LIN {X 0,Y 493.149,Z 1087.969,A -85,B 0,C 180,E1 23459.51,E2 23459.51} C_VEL
LIN {X 0,Y 495.56,Z 1076.918,A -85,B 0,C 180,E1 23456.854,E2 23456.854} C_VEL
LIN {X 0,Y 498.205,Z 1065.994,A -85,B 0,C 180,E1 23454.549,E2 23454.549} C_VEL
LIN {X 0,Y 501.969,Z 1051.472,A -85,B 0,C 180,E1 23451.868,E2 23451.868} C_VEL
LIN {X 0,Y 505.85,Z 1036.884,A -85,B 0,C 180,E1 23449.554,E2 23449.554} C_VEL
LIN {X 0,Y 509.727,Z 1022.712,A -85,B 0,C 180,E1 23447.563,E2 23447.563} C_VEL
LIN {X 0,Y 514.746,Z 1004.544,A -85,B 0,C 180,E1 23445.313,E2 23445.313} C_VEL
LIN {X 0,Y 519.682,Z 985.954,A -85,B 0,C 180,E1 23443.342,E2 23443.342} C_VEL
LIN {X 0,Y 524.249,Z 968.384,A -85,B 0,C 180,E1 23441.705,E2 23441.705} C_VEL
LIN {X 0,Y 529.619,Z 946.851,A -85,B 0,C 180,E1 23439.961,E2 23439.961} C_VEL
LIN {X 0,Y 534.306,Z 926.179,A -85,B 0,C 180,E1 23438.536,E2 23438.536} C_VEL
LIN {X 0,Y 538.281,Z 907.27,A -85,B 0,C 180,E1 23437.404,E2 23437.404} C_VEL
LIN {X 0,Y 542.76,Z 883.992,A -85,B 0,C 180,E1 23436.209,E2 23436.209} C_VEL
LIN {X 0,Y 546.654,Z 859.966,A -85,B 0,C 180,E1 23435.202,E2 23435.202} C_VEL
LIN {X 0,Y 549.579,Z 838.792,A -85,B 0,C 180,E1 23434.467,E2 23434.467} C_VEL
LIN {X 0,Y 552.455,Z 813.851,A -85,B 0,C 180,E1 23433.776,E2 23433.776} C_VEL
LIN {X 0,Y 554.553,Z 787.811,A -85,B 0,C 180,E1 23433.255,E2 23433.255} C_VEL
LIN {X 0,Y 565.206,Z 561.829,A -85,B 0,C 180,E1 23429.871,E2 23429.871} C_VEL
LIN {X 0,Y 571.63,Z 430.73,A -85,B 0,C 180,E1 23427.899,E2 23427.899} C_VEL
LIN {X 0,Y 561.962,Z 416.011,A -85,B 0,C 180,E1 23425.873,E2 23425.873} C_VEL
LIN {X 0,Y 552.616,Z 402.576,A -85,B 0,C 180,E1 23423.712,E2 23423.712} C_VEL
LIN {X 0,Y 543.559,Z 390.444,A -85,B 0,C 180,E1 23421.388,E2 23421.388} C_VEL
LIN {X 0,Y 535.724,Z 380.439,A -85,B 0,C 180,E1 23419.121,E2 23419.121} C_VEL
LIN {X 0,Y 531.614,Z 375.29,A -85,B 0,C 180,E1 23417.797,E2 23417.797} C_VEL
LIN {X 0,Y 527.184,Z 369.759,A -85,B 0,C 180,E1 23416.246,E2 23416.246} C_VEL
LIN {X 0,Y 522.155,Z 363.819,A -85,B 0,C 180,E1 23414.302,E2 23414.302} C_VEL
LIN {X 0,Y 517.658,Z 358.56,A -85,B 0,C 180,E1 23412.324,E2 23412.324} C_VEL
LIN {X 0,Y 512.757,Z 352.887,A -85,B 0,C 180,E1 23409.768,E2 23409.768} C_VEL
LIN {X 0,Y 508.771,Z 348.402,A -85,B 0,C 180,E1 23407.056,E2 23407.056} C_VEL
LIN {X 0,Y 508.042,Z 346.896,A -85,B 0,C 180,E1 23405.987,E2 23405.987} C_VEL
LIN {X 0,Y 505.565,Z 343.176,A -85,B 0,C 180,E1 23400.34,E2 23400.34} C_VEL
LIN {X 0,Y 505.432,Z 342.683,A -85,B 0,C 180,E1 23397.165,E2 23397.165} C_VEL
LIN {X 0,Y 505.943,Z 343.954,A -85,B 0,C 180,E1 23393.988,E2 23393.988} C_VEL
LIN {X 0,Y 508.736,Z 347.633,A -85,B 0,C 180,E1 23389.124,E2 23389.124} C_VEL
LIN {X 0,Y 510.625,Z 350.855,A -85,B 0,C 180,E1 23387.331,E2 23387.331} C_VEL
LIN {X 0,Y 514.02,Z 354.154,A -85,B 0,C 180,E1 23385.352,E2 23385.352} C_VEL
LIN {X 0,Y 519.518,Z 360.565,A -85,B 0,C 180,E1 23382.643,E2 23382.643} C_VEL
LIN {X 0,Y 524.302,Z 366.111,A -85,B 0,C 180,E1 23380.649,E2 23380.649} C_VEL
LIN {X 0,Y 528.297,Z 370.821,A -85,B 0,C 180,E1 23379.156,E2 23379.156} C_VEL
LIN {X 0,Y 534.627,Z 378.837,A -85,B 0,C 180,E1 23377.019,E2 23377.019} C_VEL
LIN {X 0,Y 541.875,Z 388.004,A -85,B 0,C 180,E1 23374.887,E2 23374.887} C_VEL
LIN {X 0,Y 549.446,Z 397.959,A -85,B 0,C 180,E1 23372.879,E2 23372.879} C_VEL
LIN {X 0,Y 559.137,Z 411.552,A -85,B 0,C 180,E1 23370.572,E2 23370.572} C_VEL
LIN {X 0,Y 568.555,Z 425.718,A -85,B 0,C 180,E1 23368.541,E2 23368.541} C_VEL
LIN {X 0,Y 574.364,Z 435.478,A -85,B 0,C 180,E1 23367.361,E2 23367.361} C_VEL
LIN {X 0,Y 564.405,Z 645.919,A -85,B 0,C 180,E1 23364.13,E2 23364.13} C_VEL
LIN {X 0,Y 556.556,Z 821.444,A -85,B 0,C 180,E1 23361.46,E2 23361.46} C_VEL
LIN {X 0,Y 554.253,Z 849.077,A -85,B 0,C 180,E1 23360.931,E2 23360.931} C_VEL
LIN {X 0,Y 551.182,Z 874.995,A -85,B 0,C 180,E1 23360.252,E2 23360.252} C_VEL
LIN {X 0,Y 548.203,Z 896.474,A -85,B 0,C 180,E1 23359.554,E2 23359.554} C_VEL
LIN {X 0,Y 544.933,Z 917.274,A -85,B 0,C 180,E1 23358.748,E2 23358.748} C_VEL
LIN {X 0,Y 540.875,Z 940.581,A -85,B 0,C 180,E1 23357.684,E2 23357.684} C_VEL
LIN {X 0,Y 535.726,Z 966.965,A -85,B 0,C 180,E1 23356.243,E2 23356.243} C_VEL
LIN {X 0,Y 531.462,Z 987.244,A -85,B 0,C 180,E1 23354.954,E2 23354.954} C_VEL
LIN {X 0,Y 527.075,Z 1007.137,A -85,B 0,C 180,E1 23353.52,E2 23353.52} C_VEL
LIN {X 0,Y 521.899,Z 1029.99,A -85,B 0,C 180,E1 23351.652,E2 23351.652} C_VEL
LIN {X 0,Y 516.787,Z 1051.566,A -85,B 0,C 180,E1 23349.606,E2 23349.606} C_VEL
LIN {X 0,Y 512.688,Z 1068.925,A -85,B 0,C 180,E1 23347.761,E2 23347.761} C_VEL
LIN {X 0,Y 508.88,Z 1085.197,A -85,B 0,C 180,E1 23345.84,E2 23345.84} C_VEL
LIN {X 0,Y 504.662,Z 1103.524,A -85,B 0,C 180,E1 23343.421,E2 23343.421} C_VEL
LIN {X 0,Y 500.671,Z 1121.052,A -85,B 0,C 180,E1 23340.747,E2 23340.747} C_VEL
LIN {X 0,Y 497.946,Z 1133.879,A -85,B 0,C 180,E1 23338.548,E2 23338.548} C_VEL
LIN {X 0,Y 495.478,Z 1146.019,A -85,B 0,C 180,E1 23336.227,E2 23336.227} C_VEL
LIN {X 0,Y 493.194,Z 1158.493,A -85,B 0,C 180,E1 23333.54,E2 23333.54} C_VEL
LIN {X 0,Y 491.411,Z 1169.048,A -85,B 0,C 180,E1 23330.859,E2 23330.859} C_VEL
LIN {X 0,Y 489.941,Z 1178.442,A -85,B 0,C 180,E1 23327.948,E2 23327.948} C_VEL
LIN {X 0,Y 489.053,Z 1185.745,A -85,B 0,C 180,E1 23325.292,E2 23325.292} C_VEL
LIN {X 0,Y 488.48,Z 1191.567,A -85,B 0,C 180,E1 23322.772,E2 23322.772} C_VEL
LIN {X 0,Y 488.152,Z 1196.51,A -85,B 0,C 180,E1 23320.146,E2 23320.146} C_VEL
LIN {X 0,Y 487.972,Z 1200.927,A -85,B 0,C 180,E1 23317.062,E2 23317.062} C_VEL
LIN {X 0,Y 487.915,Z 1203.615,A -85,B 0,C 180,E1 23313.995,E2 23313.995} C_VEL
LIN {X 0,Y 487.912,Z 1204.735,A -85,B 0,C 180,E1 23311.409,E2 23311.409} C_VEL
LIN {X 0,Y 487.906,Z 1204.825,A -85,B 0,C 180,E1 23309.061,E2 23309.061} C_VEL
LIN {X 0,Y 487.915,Z 1203.955,A -85,B 0,C 180,E1 23306.593,E2 23306.593} C_VEL
LIN {X 0,Y 487.942,Z 1202.076,A -85,B 0,C 180,E1 23304.119,E2 23304.119} C_VEL
LIN {X 0,Y 488.027,Z 1199.188,A -85,B 0,C 180,E1 23301.636,E2 23301.636} C_VEL
LIN {X 0,Y 488.216,Z 1195.271,A -85,B 0,C 180,E1 23299.14,E2 23299.14} C_VEL
LIN {X 0,Y 488.681,Z 1189.532,A -85,B 0,C 180,E1 23296.271,E2 23296.271} C_VEL
LIN {X 0,Y 489.58,Z 1181.265,A -85,B 0,C 180,E1 23293.02,E2 23293.02} C_VEL
LIN {X 0,Y 490.735,Z 1173.099,A -85,B 0,C 180,E1 23290.356,E2 23290.356} C_VEL
LIN {X 0,Y 492.077,Z 1164.967,A -85,B 0,C 180,E1 23288.045,E2 23288.045} C_VEL
LIN {X 0,Y 493.665,Z 1155.796,A -85,B 0,C 180,E1 23285.85,E2 23285.85} C_VEL
LIN {X 0,Y 495.728,Z 1144.888,A -85,B 0,C 180,E1 23283.529,E2 23283.529} C_VEL
LIN {X 0,Y 498.377,Z 1132.01,A -85,B 0,C 180,E1 23281.086,E2 23281.086} C_VEL
LIN {X 0,Y 502.265,Z 1114.42,A -85,B 0,C 180,E1 23278.161,E2 23278.161} C_VEL
LIN {X 0,Y 505.899,Z 1098.541,A -85,B 0,C 180,E1 23275.855,E2 23275.855} C_VEL
LIN {X 0,Y 509.534,Z 1083.124,A -85,B 0,C 180,E1 23273.848,E2 23273.848} C_VEL
LIN {X 0,Y 513.567,Z 1066.164,A -85,B 0,C 180,E1 23271.866,E2 23271.866} C_VEL
LIN {X 0,Y 518.894,Z 1043.729,A -85,B 0,C 180,E1 23269.566,E2 23269.566} C_VEL
LIN {X 0,Y 523.308,Z 1024.462,A -85,B 0,C 180,E1 23267.847,E2 23267.847} C_VEL
LIN {X 0,Y 527.446,Z 1005.817,A -85,B 0,C 180,E1 23266.369,E2 23266.369} C_VEL
LIN {X 0,Y 531.6,Z 986.265,A -85,B 0,C 180,E1 23264.993,E2 23264.993} C_VEL
LIN {X 0,Y 536.616,Z 961.242,A -85,B 0,C 180,E1 23263.462,E2 23263.462} C_VEL
LIN {X 0,Y 540.86,Z 937.419,A -85,B 0,C 180,E1 23262.236,E2 23262.236} C_VEL
LIN {X 0,Y 544.215,Z 916.811,A -85,B 0,C 180,E1 23261.325,E2 23261.325} C_VEL
LIN {X 0,Y 547.287,Z 895.889,A -85,B 0,C 180,E1 23260.536,E2 23260.536} C_VEL
LIN {X 0,Y 550.407,Z 871.646,A -85,B 0,C 180,E1 23259.775,E2 23259.775} C_VEL
LIN {X 0,Y 553.269,Z 843.484,A -85,B 0,C 180,E1 23259.097,E2 23259.097} C_VEL
LIN {X 0,Y 554.958,Z 820.18,A -85,B 0,C 180,E1 23258.674,E2 23258.674} C_VEL
LIN {X 0,Y 562.927,Z 611.986,A -85,B 0,C 180,E1 23255.596,E2 23255.596} C_VEL
LIN {X 0,Y 569.954,Z 434.455,A -85,B 0,C 180,E1 23252.946,E2 23252.946} C_VEL
LIN {X 0,Y 553.295,Z 409.736,A -85,B 0,C 180,E1 23250.158,E2 23250.158} C_VEL
LIN {X 0,Y 539.586,Z 390.209,A -85,B 0,C 180,E1 23247.628,E2 23247.628} C_VEL
LIN {X 0,Y 527.933,Z 374.572,A -85,B 0,C 180,E1 23245.253,E2 23245.253} C_VEL
LIN {X 0,Y 517.455,Z 360.976,A -85,B 0,C 180,E1 23242.915,E2 23242.915} C_VEL
LIN {X 0,Y 511.897,Z 354.221,A -85,B 0,C 180,E1 23241.575,E2 23241.575} C_VEL
LIN {X 0,Y 507.878,Z 349.051,A -85,B 0,C 180,E1 23240.514,E2 23240.514} C_VEL
LIN {X 0,Y 505.11,Z 344.247,A -85,B 0,C 180,E1 23239.184,E2 23239.184} C_VEL
LIN {X 0,Y 502.34,Z 339.33,A -85,B 0,C 180,E1 23237.731,E2 23237.731} C_VEL
LIN {X 0,Y 500.084,Z 335.455,A -85,B 0,C 180,E1 23236.494,E2 23236.494} C_VEL
LIN {X 0,Y 499.057,Z 333.831,A -85,B 0,C 180,E1 23235.932,E2 23235.932} C_VEL
LIN {X 0,Y 496.972,Z 330.249,A -85,B 0,C 180,E1 23234.685,E2 23234.685} C_VEL
LIN {X 0,Y 496.045,Z 328.722,A -85,B 0,C 180,E1 23234.117,E2 23234.117} C_VEL
LIN {X 0,Y 493.83,Z 325.381,A -85,B 0,C 180,E1 23232.75,E2 23232.75} C_VEL
LIN {X 0,Y 492.938,Z 323.506,A -85,B 0,C 180,E1 23232.06,E2 23232.06} C_VEL
LIN {X 0,Y 490.401,Z 319.891,A -85,B 0,C 180,E1 23230.336,E2 23230.336} C_VEL
LIN {X 0,Y 490.011,Z 318.347,A -85,B 0,C 180,E1 23229.632,E2 23229.632} C_VEL
LIN {X 0,Y 489.975,Z 318.197,A -85,B 0,C 180,E1 23226.327,E2 23226.327} C_VEL
LIN {X 0,Y 489.984,Z 318.197,A -85,B 0,C 180,E1 23222.69,E2 23222.69} C_VEL
LIN {X 0,Y 489.988,Z 318.196,A -85,B 0,C 180,E1 23219.11,E2 23219.11} C_VEL
LIN {X 0,Y 489.979,Z 318.198,A -85,B 0,C 180,E1 23215.552,E2 23215.552} C_VEL
LIN {X 0,Y 489.968,Z 318.2,A -85,B 0,C 180,E1 23212.023,E2 23212.023} C_VEL
LIN {X 0,Y 489.987,Z 318.199,A -85,B 0,C 180,E1 23208.464,E2 23208.464} C_VEL
LIN {X 0,Y 489.996,Z 318.196,A -85,B 0,C 180,E1 23204.835,E2 23204.835} C_VEL
LIN {X 0,Y 489.973,Z 318.196,A -85,B 0,C 180,E1 23201.236,E2 23201.236} C_VEL
LIN {X 0,Y 489.962,Z 318.184,A -85,B 0,C 180,E1 23197.692,E2 23197.692} C_VEL
LIN {X 0,Y 490.031,Z 318.559,A -85,B 0,C 180,E1 23195.915,E2 23195.915} C_VEL
LIN {X 0,Y 491.731,Z 322.184,A -85,B 0,C 180,E1 23194.334,E2 23194.334} C_VEL
LIN {X 0,Y 493.389,Z 324.398,A -85,B 0,C 180,E1 23193.263,E2 23193.263} C_VEL
LIN {X 0,Y 495.592,Z 328.394,A -85,B 0,C 180,E1 23191.697,E2 23191.697} C_VEL
LIN {X 0,Y 496.572,Z 329.857,A -85,B 0,C 180,E1 23191.101,E2 23191.101} C_VEL
LIN {X 0,Y 498.866,Z 333.836,A -85,B 0,C 180,E1 23189.663,E2 23189.663} C_VEL
LIN {X 0,Y 502.443,Z 340.404,A -85,B 0,C 180,E1 23187.539,E2 23187.539} C_VEL
LIN {X 0,Y 505.203,Z 345.524,A -85,B 0,C 180,E1 23186.022,E2 23186.022} C_VEL
LIN {X 0,Y 507.222,Z 348.663,A -85,B 0,C 180,E1 23185.201,E2 23185.201} C_VEL
LIN {X 0,Y 513.433,Z 356.368,A -85,B 0,C 180,E1 23183.629,E2 23183.629} C_VEL
LIN {X 0,Y 523.089,Z 368.663,A -85,B 0,C 180,E1 23181.383,E2 23181.383} C_VEL
LIN {X 0,Y 533.138,Z 382.053,A -85,B 0,C 180,E1 23179.259,E2 23179.259} C_VEL
LIN {X 0,Y 545.23,Z 398.991,A -85,B 0,C 180,E1 23176.912,E2 23176.912} C_VEL
LIN {X 0,Y 559.529,Z 420.202,A -85,B 0,C 180,E1 23174.39,E2 23174.39} C_VEL
LIN {X 0,Y 564.66,Z 428.424,A -85,B 0,C 180,E1 23173.534,E2 23173.534} C_VEL
LIN {X 0,Y 555.474,Z 654.275,A -85,B 0,C 180,E1 23170.226,E2 23170.226} C_VEL
LIN {X 0,Y 550.131,Z 787.111,A -85,B 0,C 180,E1 23168.273,E2 23168.273} C_VEL
LIN {X 0,Y 548.159,Z 813.65,A -85,B 0,C 180,E1 23167.744,E2 23167.744} C_VEL
LIN {X 0,Y 545.611,Z 837.887,A -85,B 0,C 180,E1 23167.078,E2 23167.078} C_VEL
LIN {X 0,Y 543.174,Z 857.409,A -85,B 0,C 180,E1 23166.414,E2 23166.414} C_VEL
LIN {X 0,Y 541.449,Z 864.935,A -85,B 0,C 180,E1 23166.216,E2 23166.216} C_VEL
LIN {X 0,Y 534.335,Z 883.517,A -85,B 0,C 180,E1 23165.889,E2 23165.889} C_VEL
LIN {X 0,Y 532.422,Z 890.42,A -85,B 0,C 180,E1 23165.628,E2 23165.628} C_VEL
LIN {X 0,Y 528.887,Z 909.703,A -85,B 0,C 180,E1 23164.617,E2 23164.617} C_VEL
LIN {X 0,Y 524.361,Z 932.228,A -85,B 0,C 180,E1 23163.244,E2 23163.244} C_VEL
LIN {X 0,Y 519.531,Z 953.612,A -85,B 0,C 180,E1 23161.695,E2 23161.695} C_VEL
LIN {X 0,Y 515.319,Z 971.28,A -85,B 0,C 180,E1 23160.232,E2 23160.232} C_VEL
LIN {X 0,Y 510.276,Z 991.608,A -85,B 0,C 180,E1 23158.306,E2 23158.306} C_VEL
LIN {X 0,Y 505.499,Z 1009.737,A -85,B 0,C 180,E1 23156.299,E2 23156.299} C_VEL
LIN {X 0,Y 501.644,Z 1024.173,A -85,B 0,C 180,E1 23154.493,E2 23154.493} C_VEL
LIN {X 0,Y 497.358,Z 1040.344,A -85,B 0,C 180,E1 23152.206,E2 23152.206} C_VEL
LIN {X 0,Y 493.255,Z 1055.784,A -85,B 0,C 180,E1 23149.663,E2 23149.663} C_VEL
LIN {X 0,Y 490.261,Z 1067.568,A -85,B 0,C 180,E1 23147.445,E2 23147.445} C_VEL
LIN {X 0,Y 487.453,Z 1079.24,A -85,B 0,C 180,E1 23144.951,E2 23144.951} C_VEL
LIN {X 0,Y 484.785,Z 1091.351,A -85,B 0,C 180,E1 23141.902,E2 23141.902} C_VEL
LIN {X 0,Y 483.145,Z 1099.766,A -85,B 0,C 180,E1 23139.409,E2 23139.409} C_VEL
LIN {X 0,Y 481.86,Z 1107.651,A -85,B 0,C 180,E1 23136.673,E2 23136.673} C_VEL
LIN {X 0,Y 480.875,Z 1115.108,A -85,B 0,C 180,E1 23133.457,E2 23133.457} C_VEL
LIN {X 0,Y 480.406,Z 1119.686,A -85,B 0,C 180,E1 23130.954,E2 23130.954} C_VEL
LIN {X 0,Y 480.182,Z 1123.237,A -85,B 0,C 180,E1 23128.449,E2 23128.449} C_VEL
LIN {X 0,Y 480.051,Z 1126.112,A -85,B 0,C 180,E1 23125.58,E2 23125.58} C_VEL
LIN {X 0,Y 480.017,Z 1127.597,A -85,B 0,C 180,E1 23122.536,E2 23122.536} C_VEL
LIN {X 0,Y 480.009,Z 1127.73,A -85,B 0,C 180,E1 23120.044,E2 23120.044} C_VEL
LIN {X 0,Y 480.042,Z 1126.911,A -85,B 0,C 180,E1 23117.612,E2 23117.612} C_VEL
LIN {X 0,Y 480.092,Z 1125.029,A -85,B 0,C 180,E1 23115.034,E2 23115.034} C_VEL
LIN {X 0,Y 480.33,Z 1121.374,A -85,B 0,C 180,E1 23111.931,E2 23111.931} C_VEL
LIN {X 0,Y 480.725,Z 1116.685,A -85,B 0,C 180,E1 23109.166,E2 23109.166} C_VEL
LIN {X 0,Y 481.392,Z 1111.294,A -85,B 0,C 180,E1 23106.627,E2 23106.627} C_VEL
LIN {X 0,Y 482.54,Z 1104.025,A -85,B 0,C 180,E1 23103.798,E2 23103.798} C_VEL
LIN {X 0,Y 484.362,Z 1094.295,A -85,B 0,C 180,E1 23100.71,E2 23100.71} C_VEL
LIN {X 0,Y 486.355,Z 1085.178,A -85,B 0,C 180,E1 23098.245,E2 23098.245} C_VEL
LIN {X 0,Y 489.044,Z 1074.172,A -85,B 0,C 180,E1 23095.647,E2 23095.647} C_VEL
LIN {X 0,Y 492.766,Z 1060.042,A -85,B 0,C 180,E1 23092.795,E2 23092.795} C_VEL
LIN {X 0,Y 496.209,Z 1047.557,A -85,B 0,C 180,E1 23090.6,E2 23090.6} C_VEL
LIN {X 0,Y 500.308,Z 1033.218,A -85,B 0,C 180,E1 23088.371,E2 23088.371} C_VEL
LIN {X 0,Y 505.662,Z 1014.624,A -85,B 0,C 180,E1 23085.873,E2 23085.873} C_VEL
LIN {X 0,Y 509.914,Z 999.653,A -85,B 0,C 180,E1 23084.117,E2 23084.117} C_VEL
LIN {X 0,Y 514.514,Z 983.146,A -85,B 0,C 180,E1 23082.4,E2 23082.4} C_VEL
LIN {X 0,Y 520.076,Z 962.549,A -85,B 0,C 180,E1 23080.529,E2 23080.529} C_VEL
LIN {X 0,Y 525.106,Z 942.324,A -85,B 0,C 180,E1 23078.962,E2 23078.962} C_VEL
LIN {X 0,Y 529.206,Z 924.828,A -85,B 0,C 180,E1 23077.776,E2 23077.776} C_VEL
LIN {X 0,Y 533.347,Z 905.742,A -85,B 0,C 180,E1 23076.643,E2 23076.643} C_VEL
LIN {X 0,Y 538.141,Z 881.083,A -85,B 0,C 180,E1 23075.405,E2 23075.405} C_VEL
LIN {X 0,Y 541.68,Z 859.732,A -85,B 0,C 180,E1 23074.52,E2 23074.52} C_VEL
LIN {X 0,Y 544.703,Z 838.45,A -85,B 0,C 180,E1 23073.786,E2 23073.786} C_VEL
LIN {X 0,Y 547.724,Z 812.789,A -85,B 0,C 180,E1 23073.081,E2 23073.081} C_VEL
LIN {X 0,Y 549.775,Z 787.528,A -85,B 0,C 180,E1 23072.582,E2 23072.582} C_VEL
LIN {X 0,Y 561.031,Z 557.477,A -85,B 0,C 180,E1 23069.121,E2 23069.121} C_VEL
LIN {X 0,Y 567.259,Z 435.24,A -85,B 0,C 180,E1 23067.277,E2 23067.277} C_VEL
LIN {X 0,Y 558.135,Z 421.099,A -85,B 0,C 180,E1 23065.295,E2 23065.295} C_VEL
LIN {X 0,Y 548.312,Z 407.108,A -85,B 0,C 180,E1 23062.942,E2 23062.942} C_VEL
LIN {X 0,Y 540.587,Z 396.703,A -85,B 0,C 180,E1 23060.887,E2 23060.887} C_VEL
LIN {X 0,Y 533.593,Z 387.597,A -85,B 0,C 180,E1 23058.803,E2 23058.803} C_VEL
LIN {X 0,Y 529.702,Z 382.655,A -85,B 0,C 180,E1 23057.523,E2 23057.523} C_VEL
LIN {X 0,Y 525.337,Z 377.159,A -85,B 0,C 180,E1 23055.964,E2 23055.964} C_VEL
LIN {X 0,Y 520.538,Z 371.373,A -85,B 0,C 180,E1 23054.069,E2 23054.069} C_VEL
LIN {X 0,Y 516.098,Z 366.142,A -85,B 0,C 180,E1 23052.078,E2 23052.078} C_VEL
LIN {X 0,Y 511.399,Z 360.607,A -85,B 0,C 180,E1 23049.567,E2 23049.567} C_VEL
LIN {X 0,Y 507.466,Z 356.08,A -85,B 0,C 180,E1 23046.846,E2 23046.846} C_VEL
LIN {X 0,Y 506.221,Z 354.581,A -85,B 0,C 180,E1 23045.782,E2 23045.782} C_VEL
LIN {X 0,Y 502.063,Z 350.235,A -85,B 0,C 180,E1 23039.886,E2 23039.886} C_VEL
LIN {X 0,Y 501.879,Z 349.869,A -85,B 0,C 180,E1 23037.031,E2 23037.031} C_VEL
LIN {X 0,Y 502.965,Z 351.467,A -85,B 0,C 180,E1 23033.837,E2 23033.837} C_VEL
LIN {X 0,Y 507.148,Z 355.467,A -85,B 0,C 180,E1 23029.205,E2 23029.205} C_VEL
LIN {X 0,Y 511.664,Z 360.798,A -85,B 0,C 180,E1 23026.092,E2 23026.092} C_VEL
LIN {X 0,Y 514.654,Z 364.49,A -85,B 0,C 180,E1 23024.448,E2 23024.448} C_VEL
LIN {X 0,Y 517.936,Z 368.114,A -85,B 0,C 180,E1 23022.878,E2 23022.878} C_VEL
LIN {X 0,Y 522.709,Z 373.78,A -85,B 0,C 180,E1 23020.849,E2 23020.849} C_VEL
LIN {X 0,Y 527.586,Z 379.753,A -85,B 0,C 180,E1 23019.01,E2 23019.01} C_VEL
LIN {X 0,Y 532.838,Z 386.422,A -85,B 0,C 180,E1 23017.23,E2 23017.23} C_VEL
LIN {X 0,Y 539.82,Z 395.404,A -85,B 0,C 180,E1 23015.136,E2 23015.136} C_VEL
LIN {X 0,Y 547.118,Z 405.126,A -85,B 0,C 180,E1 23013.166,E2 23013.166} C_VEL
LIN {X 0,Y 556.468,Z 418.446,A -85,B 0,C 180,E1 23010.889,E2 23010.889} C_VEL
LIN {X 0,Y 566.323,Z 433.447,A -85,B 0,C 180,E1 23008.729,E2 23008.729} C_VEL
LIN {X 0,Y 569.9,Z 439.665,A -85,B 0,C 180,E1 23007.98,E2 23007.98} C_VEL
LIN {X 0,Y 559.578,Z 649.32,A -85,B 0,C 180,E1 23004.745,E2 23004.745} C_VEL
LIN {X 0,Y 551.576,Z 820.917,A -85,B 0,C 180,E1 23002.118,E2 23002.118} C_VEL
LIN {X 0,Y 549.197,Z 848.626,A -85,B 0,C 180,E1 23001.585,E2 23001.585} C_VEL
LIN {X 0,Y 546.027,Z 874.538,A -85,B 0,C 180,E1 23000.907,E2 23000.907} C_VEL
LIN {X 0,Y 542.938,Z 895.975,A -85,B 0,C 180,E1 23000.21,E2 23000.21} C_VEL
LIN {X 0,Y 539.664,Z 916.061,A -85,B 0,C 180,E1 22999.431,E2 22999.431} C_VEL
LIN {X 0,Y 535.762,Z 937.687,A -85,B 0,C 180,E1 22998.449,E2 22998.449} C_VEL
LIN {X 0,Y 530.406,Z 964.478,A -85,B 0,C 180,E1 22997.005,E2 22997.005} C_VEL
LIN {X 0,Y 525.551,Z 986.636,A -85,B 0,C 180,E1 22995.593,E2 22995.593} C_VEL
LIN {X 0,Y 521.003,Z 1006.41,A -85,B 0,C 180,E1 22994.158,E2 22994.158} C_VEL
LIN {X 0,Y 515.614,Z 1029.058,A -85,B 0,C 180,E1 22992.29,E2 22992.29} C_VEL
LIN {X 0,Y 510.083,Z 1051.281,A -85,B 0,C 180,E1 22990.158,E2 22990.158} C_VEL
LIN {X 0,Y 505.808,Z 1068.507,A -85,B 0,C 180,E1 22988.298,E2 22988.298} C_VEL
LIN {X 0,Y 501.484,Z 1086.179,A -85,B 0,C 180,E1 22986.169,E2 22986.169} C_VEL
LIN {X 0,Y 496.7,Z 1105.888,A -85,B 0,C 180,E1 22983.474,E2 22983.474} C_VEL
LIN {X 0,Y 493.164,Z 1120.911,A -85,B 0,C 180,E1 22981.131,E2 22981.131} C_VEL
LIN {X 0,Y 490.332,Z 1133.702,A -85,B 0,C 180,E1 22978.9,E2 22978.9} C_VEL
LIN {X 0,Y 487.769,Z 1145.806,A -85,B 0,C 180,E1 22976.543,E2 22976.543} C_VEL
LIN {X 0,Y 485.199,Z 1159.334,A -85,B 0,C 180,E1 22973.564,E2 22973.564} C_VEL
LIN {X 0,Y 483.25,Z 1170.749,A -85,B 0,C 180,E1 22970.594,E2 22970.594} C_VEL
LIN {X 0,Y 482.21,Z 1177.735,A -85,B 0,C 180,E1 22968.496,E2 22968.496} C_VEL
LIN {X 0,Y 481.205,Z 1185.136,A -85,B 0,C 180,E1 22965.795,E2 22965.795} C_VEL
LIN {X 0,Y 480.582,Z 1191.055,A -85,B 0,C 180,E1 22963.23,E2 22963.23} C_VEL
LIN {X 0,Y 480.205,Z 1195.887,A -85,B 0,C 180,E1 22960.679,E2 22960.679} C_VEL
LIN {X 0,Y 480.02,Z 1199.666,A -85,B 0,C 180,E1 22958.143,E2 22958.143} C_VEL
LIN {X 0,Y 479.935,Z 1202.529,A -85,B 0,C 180,E1 22955.499,E2 22955.499} C_VEL
LIN {X 0,Y 479.909,Z 1204.549,A -85,B 0,C 180,E1 22952.388,E2 22952.388} C_VEL
LIN {X 0,Y 479.898,Z 1204.871,A -85,B 0,C 180,E1 22949.284,E2 22949.284} C_VEL
LIN {X 0,Y 479.915,Z 1204.02,A -85,B 0,C 180,E1 22946.656,E2 22946.656} C_VEL
LIN {X 0,Y 479.942,Z 1202.187,A -85,B 0,C 180,E1 22944.141,E2 22944.141} C_VEL
LIN {X 0,Y 480.03,Z 1199.345,A -85,B 0,C 180,E1 22941.616,E2 22941.616} C_VEL
LIN {X 0,Y 480.227,Z 1195.474,A -85,B 0,C 180,E1 22939.078,E2 22939.078} C_VEL
LIN {X 0,Y 480.66,Z 1190.292,A -85,B 0,C 180,E1 22936.405,E2 22936.405} C_VEL
LIN {X 0,Y 481.54,Z 1182.564,A -85,B 0,C 180,E1 22933.185,E2 22933.185} C_VEL
LIN {X 0,Y 482.736,Z 1174.205,A -85,B 0,C 180,E1 22930.395,E2 22930.395} C_VEL
LIN {X 0,Y 484.234,Z 1164.767,A -85,B 0,C 180,E1 22927.799,E2 22927.799} C_VEL
LIN {X 0,Y 486.001,Z 1154.944,A -85,B 0,C 180,E1 22925.418,E2 22925.418} C_VEL
LIN {X 0,Y 488.291,Z 1143.561,A -85,B 0,C 180,E1 22922.97,E2 22922.97} C_VEL
LIN {X 0,Y 491.398,Z 1129.213,A -85,B 0,C 180,E1 22920.233,E2 22920.233} C_VEL
LIN {X 0,Y 495.397,Z 1111.974,A -85,B 0,C 180,E1 22917.392,E2 22917.392} C_VEL
LIN {X 0,Y 498.899,Z 1097.366,A -85,B 0,C 180,E1 22915.258,E2 22915.258} C_VEL
LIN {X 0,Y 502.721,Z 1081.882,A -85,B 0,C 180,E1 22913.226,E2 22913.226} C_VEL
LIN {X 0,Y 507.116,Z 1064.206,A -85,B 0,C 180,E1 22911.154,E2 22911.154} C_VEL
LIN {X 0,Y 512.712,Z 1041.417,A -85,B 0,C 180,E1 22908.832,E2 22908.832} C_VEL
LIN {X 0,Y 517.1,Z 1022.93,A -85,B 0,C 180,E1 22907.183,E2 22907.183} C_VEL
LIN {X 0,Y 521.321,Z 1004.538,A -85,B 0,C 180,E1 22905.723,E2 22905.723} C_VEL
LIN {X 0,Y 525.844,Z 983.937,A -85,B 0,C 180,E1 22904.276,E2 22904.276} C_VEL
LIN {X 0,Y 531.213,Z 957.473,A -85,B 0,C 180,E1 22902.685,E2 22902.685} C_VEL
LIN {X 0,Y 535.121,Z 936.125,A -85,B 0,C 180,E1 22901.591,E2 22901.591} C_VEL
LIN {X 0,Y 538.524,Z 915.852,A -85,B 0,C 180,E1 22900.696,E2 22900.696} C_VEL
LIN {X 0,Y 541.75,Z 894.371,A -85,B 0,C 180,E1 22899.887,E2 22899.887} C_VEL
LIN {X 0,Y 545.265,Z 867.462,A -85,B 0,C 180,E1 22899.057,E2 22899.057} C_VEL
LIN {X 0,Y 547.902,Z 841.288,A -85,B 0,C 180,E1 22898.449,E2 22898.449} C_VEL
LIN {X 0,Y 549.55,Z 818.677,A -85,B 0,C 180,E1 22898.042,E2 22898.042} C_VEL
LIN {X 0,Y 558.019,Z 604.996,A -85,B 0,C 180,E1 22894.865,E2 22894.865} C_VEL
LIN {X 0,Y 564.797,Z 438.419,A -85,B 0,C 180,E1 22892.355,E2 22892.355} C_VEL
LIN {X 0,Y 548.205,Z 413.645,A -85,B 0,C 180,E1 22889.503,E2 22889.503} C_VEL
LIN {X 0,Y 535.093,Z 394.942,A -85,B 0,C 180,E1 22887.006,E2 22887.006} C_VEL
LIN {X 0,Y 524.293,Z 380.36,A -85,B 0,C 180,E1 22884.747,E2 22884.747} C_VEL
LIN {X 0,Y 514.402,Z 367.495,A -85,B 0,C 180,E1 22882.485,E2 22882.485} C_VEL
LIN {X 0,Y 509.447,Z 361.312,A -85,B 0,C 180,E1 22881.261,E2 22881.261} C_VEL
LIN {X 0,Y 505.09,Z 355.837,A -85,B 0,C 180,E1 22880.118,E2 22880.118} C_VEL
LIN {X 0,Y 499.482,Z 349.183,A -85,B 0,C 180,E1 22878.56,E2 22878.56} C_VEL
LIN {X 0,Y 497.58,Z 345.614,A -85,B 0,C 180,E1 22877.543,E2 22877.543} C_VEL
LIN {X 0,Y 495.238,Z 341.26,A -85,B 0,C 180,E1 22876.178,E2 22876.178} C_VEL
LIN {X 0,Y 492.464,Z 336.882,A -85,B 0,C 180,E1 22874.582,E2 22874.582} C_VEL
LIN {X 0,Y 491.577,Z 335.301,A -85,B 0,C 180,E1 22874.008,E2 22874.008} C_VEL
LIN {X 0,Y 489.376,Z 331.972,A -85,B 0,C 180,E1 22872.628,E2 22872.628} C_VEL
LIN {X 0,Y 488.494,Z 330.101,A -85,B 0,C 180,E1 22871.931,E2 22871.931} C_VEL
LIN {X 0,Y 486.006,Z 326.464,A -85,B 0,C 180,E1 22870.191,E2 22870.191} C_VEL
LIN {X 0,Y 485.115,Z 324.567,A -85,B 0,C 180,E1 22869.371,E2 22869.371} C_VEL
LIN {X 0,Y 482.51,Z 321.013,A -85,B 0,C 180,E1 22867.262,E2 22867.262} C_VEL
LIN {X 0,Y 482.054,Z 319.32,A -85,B 0,C 180,E1 22866.312,E2 22866.312} C_VEL
LIN {X 0,Y 482.046,Z 319.187,A -85,B 0,C 180,E1 22862.735,E2 22862.735} C_VEL
LIN {X 0,Y 482.051,Z 319.186,A -85,B 0,C 180,E1 22859.168,E2 22859.168} C_VEL
LIN {X 0,Y 482.043,Z 319.184,A -85,B 0,C 180,E1 22855.479,E2 22855.479} C_VEL
LIN {X 0,Y 482.028,Z 319.187,A -85,B 0,C 180,E1 22851.891,E2 22851.891} C_VEL
LIN {X 0,Y 482.04,Z 319.183,A -85,B 0,C 180,E1 22848.245,E2 22848.245} C_VEL
LIN {X 0,Y 482.054,Z 319.178,A -85,B 0,C 180,E1 22844.603,E2 22844.603} C_VEL
LIN {X 0,Y 482.046,Z 319.177,A -85,B 0,C 180,E1 22840.994,E2 22840.994} C_VEL
LIN {X 0,Y 482.092,Z 319.544,A -85,B 0,C 180,E1 22839.148,E2 22839.148} C_VEL
LIN {X 0,Y 483.873,Z 323.339,A -85,B 0,C 180,E1 22837.139,E2 22837.139} C_VEL
LIN {X 0,Y 485.499,Z 325.314,A -85,B 0,C 180,E1 22835.934,E2 22835.934} C_VEL
LIN {X 0,Y 487.635,Z 329.224,A -85,B 0,C 180,E1 22834.176,E2 22834.176} C_VEL
LIN {X 0,Y 488.815,Z 330.954,A -85,B 0,C 180,E1 22833.364,E2 22833.364} C_VEL
LIN {X 0,Y 490.962,Z 334.863,A -85,B 0,C 180,E1 22831.804,E2 22831.804} C_VEL
LIN {X 0,Y 491.946,Z 336.485,A -85,B 0,C 180,E1 22831.162,E2 22831.162} C_VEL
LIN {X 0,Y 494.759,Z 341.394,A -85,B 0,C 180,E1 22829.384,E2 22829.384} C_VEL
LIN {X 0,Y 497.588,Z 346.645,A -85,B 0,C 180,E1 22827.688,E2 22827.688} C_VEL
LIN {X 0,Y 500.354,Z 350.433,A -85,B 0,C 180,E1 22826.732,E2 22826.732} C_VEL
LIN {X 0,Y 506.504,Z 357.974,A -85,B 0,C 180,E1 22825.076,E2 22825.076} C_VEL
LIN {X 0,Y 510.956,Z 363.442,A -85,B 0,C 180,E1 22823.946,E2 22823.946} C_VEL
LIN {X 0,Y 520.615,Z 375.882,A -85,B 0,C 180,E1 22821.658,E2 22821.658} C_VEL
LIN {X 0,Y 530.812,Z 389.685,A -85,B 0,C 180,E1 22819.467,E2 22819.467} C_VEL
LIN {X 0,Y 542.071,Z 405.63,A -85,B 0,C 180,E1 22817.249,E2 22817.249} C_VEL
LIN {X 0,Y 555.898,Z 426.345,A -85,B 0,C 180,E1 22814.762,E2 22814.762} C_VEL
LIN {X 0,Y 559.618,Z 432.343,A -85,B 0,C 180,E1 22814.126,E2 22814.126} C_VEL
LIN {X 0,Y 550.133,Z 657.447,A -85,B 0,C 180,E1 22810.812,E2 22810.812} C_VEL
LIN {X 0,Y 544.723,Z 787.47,A -85,B 0,C 180,E1 22808.889,E2 22808.889} C_VEL
LIN {X 0,Y 542.7,Z 813.954,A -85,B 0,C 180,E1 22808.359,E2 22808.359} C_VEL
LIN {X 0,Y 540.064,Z 838.316,A -85,B 0,C 180,E1 22807.687,E2 22807.687} C_VEL
LIN {X 0,Y 537.371,Z 859.114,A -85,B 0,C 180,E1 22806.974,E2 22806.974} C_VEL
LIN {X 0,Y 533.889,Z 882.265,A -85,B 0,C 180,E1 22806.019,E2 22806.019} C_VEL
LIN {X 0,Y 532.422,Z 890.42,A -85,B 0,C 180,E1 22805.628,E2 22805.628} C_VEL
LIN {X 0,Y 530.469,Z 897.664,A -85,B 0,C 180,E1 22805.352,E2 22805.352} C_VEL
LIN {X 0,Y 522.747,Z 915.523,A -85,B 0,C 180,E1 22804.842,E2 22804.842} C_VEL
LIN {X 0,Y 520.601,Z 922.243,A -85,B 0,C 180,E1 22804.505,E2 22804.505} C_VEL
LIN {X 0,Y 516.551,Z 940.681,A -85,B 0,C 180,E1 22803.281,E2 22803.281} C_VEL
LIN {X 0,Y 512.02,Z 959.934,A -85,B 0,C 180,E1 22801.82,E2 22801.82} C_VEL
LIN {X 0,Y 506.521,Z 981.683,A -85,B 0,C 180,E1 22799.896,E2 22799.896} C_VEL
LIN {X 0,Y 502.159,Z 998.111,A -85,B 0,C 180,E1 22798.222,E2 22798.222} C_VEL
LIN {X 0,Y 497.993,Z 1013.363,A -85,B 0,C 180,E1 22796.47,E2 22796.47} C_VEL
LIN {X 0,Y 493.068,Z 1031.205,A -85,B 0,C 180,E1 22794.139,E2 22794.139} C_VEL
LIN {X 0,Y 488.856,Z 1046.218,A -85,B 0,C 180,E1 22791.854,E2 22791.854} C_VEL
LIN {X 0,Y 485.329,Z 1059.162,A -85,B 0,C 180,E1 22789.621,E2 22789.621} C_VEL
LIN {X 0,Y 481.683,Z 1073.121,A -85,B 0,C 180,E1 22786.871,E2 22786.871} C_VEL
LIN {X 0,Y 478.79,Z 1084.824,A -85,B 0,C 180,E1 22784.142,E2 22784.142} C_VEL
LIN {X 0,Y 476.76,Z 1093.813,A -85,B 0,C 180,E1 22781.737,E2 22781.737} C_VEL
LIN {X 0,Y 474.876,Z 1103.517,A -85,B 0,C 180,E1 22778.719,E2 22778.719} C_VEL
LIN {X 0,Y 473.571,Z 1111.345,A -85,B 0,C 180,E1 22775.695,E2 22775.695} C_VEL
LIN {X 0,Y 472.865,Z 1116.778,A -85,B 0,C 180,E1 22773.151,E2 22773.151} C_VEL
LIN {X 0,Y 472.403,Z 1121.549,A -85,B 0,C 180,E1 22770.364,E2 22770.364} C_VEL
LIN {X 0,Y 472.134,Z 1125.514,A -85,B 0,C 180,E1 22767.087,E2 22767.087} C_VEL
LIN {X 0,Y 472.055,Z 1127.498,A -85,B 0,C 180,E1 22764.409,E2 22764.409} C_VEL
LIN {X 0,Y 472.054,Z 1128.38,A -85,B 0,C 180,E1 22761.841,E2 22761.841} C_VEL
LIN {X 0,Y 472.045,Z 1128.204,A -85,B 0,C 180,E1 22758.887,E2 22758.887} C_VEL
LIN {X 0,Y 472.11,Z 1126.426,A -85,B 0,C 180,E1 22755.778,E2 22755.778} C_VEL
LIN {X 0,Y 472.248,Z 1123.929,A -85,B 0,C 180,E1 22753.265,E2 22753.265} C_VEL
LIN {X 0,Y 472.524,Z 1120.369,A -85,B 0,C 180,E1 22750.694,E2 22750.694} C_VEL
LIN {X 0,Y 473.167,Z 1114.863,A -85,B 0,C 180,E1 22747.644,E2 22747.644} C_VEL
LIN {X 0,Y 474.277,Z 1107.482,A -85,B 0,C 180,E1 22744.528,E2 22744.528} C_VEL
LIN {X 0,Y 475.682,Z 1100.048,A -85,B 0,C 180,E1 22741.911,E2 22741.911} C_VEL
LIN {X 0,Y 477.935,Z 1089.962,A -85,B 0,C 180,E1 22738.887,E2 22738.887} C_VEL
LIN {X 0,Y 480.821,Z 1078.315,A -85,B 0,C 180,E1 22735.987,E2 22735.987} C_VEL
LIN {X 0,Y 483.772,Z 1067.437,A -85,B 0,C 180,E1 22733.618,E2 22733.618} C_VEL
LIN {X 0,Y 487.976,Z 1052.987,A -85,B 0,C 180,E1 22730.869,E2 22730.869} C_VEL
LIN {X 0,Y 492.445,Z 1037.78,A -85,B 0,C 180,E1 22728.399,E2 22728.399} C_VEL
LIN {X 0,Y 496.778,Z 1023.413,A -85,B 0,C 180,E1 22726.342,E2 22726.342} C_VEL
LIN {X 0,Y 502.27,Z 1005.215,A -85,B 0,C 180,E1 22724.058,E2 22724.058} C_VEL
LIN {X 0,Y 507.503,Z 987.189,A -85,B 0,C 180,E1 22722.118,E2 22722.118} C_VEL
LIN {X 0,Y 512.25,Z 970.34,A -85,B 0,C 180,E1 22720.521,E2 22720.521} C_VEL
LIN {X 0,Y 517.813,Z 949.801,A -85,B 0,C 180,E1 22718.819,E2 22718.819} C_VEL
LIN {X 0,Y 523.141,Z 928.071,A -85,B 0,C 180,E1 22717.293,E2 22717.293} C_VEL
LIN {X 0,Y 527.434,Z 909.087,A -85,B 0,C 180,E1 22716.141,E2 22716.141} C_VEL
LIN {X 0,Y 531.79,Z 887.911,A -85,B 0,C 180,E1 22715.034,E2 22715.034} C_VEL
LIN {X 0,Y 536.309,Z 862.557,A -85,B 0,C 180,E1 22713.939,E2 22713.939} C_VEL
LIN {X 0,Y 539.517,Z 840.946,A -85,B 0,C 180,E1 22713.178,E2 22713.178} C_VEL
LIN {X 0,Y 542.304,Z 818.41,A -85,B 0,C 180,E1 22712.537,E2 22712.537} C_VEL
LIN {X 0,Y 544.883,Z 790.236,A -85,B 0,C 180,E1 22711.946,E2 22711.946} C_VEL
LIN {X 0,Y 549.026,Z 709.383,A -85,B 0,C 180,E1 22710.711,E2 22710.711} C_VEL
LIN {X 0,Y 561.15,Z 473.673,A -85,B 0,C 180,E1 22707.161,E2 22707.161} C_VEL
LIN {X 0,Y 562.872,Z 439.476,A -85,B 0,C 180,E1 22706.622,E2 22706.622} C_VEL
LIN {X 0,Y 554.549,Z 426.67,A -85,B 0,C 180,E1 22704.757,E2 22704.757} C_VEL
LIN {X 0,Y 545.788,Z 413.969,A -85,B 0,C 180,E1 22702.598,E2 22702.598} C_VEL
LIN {X 0,Y 538.015,Z 403.372,A -85,B 0,C 180,E1 22700.479,E2 22700.479} C_VEL
LIN {X 0,Y 531.48,Z 394.75,A -85,B 0,C 180,E1 22698.482,E2 22698.482} C_VEL
LIN {X 0,Y 527.802,Z 390.017,A -85,B 0,C 180,E1 22697.246,E2 22697.246} C_VEL
LIN {X 0,Y 523.503,Z 384.552,A -85,B 0,C 180,E1 22695.68,E2 22695.68} C_VEL
LIN {X 0,Y 518.778,Z 378.762,A -85,B 0,C 180,E1 22693.771,E2 22693.771} C_VEL
LIN {X 0,Y 514.549,Z 373.722,A -85,B 0,C 180,E1 22691.83,E2 22691.83} C_VEL
LIN {X 0,Y 510.237,Z 368.482,A -85,B 0,C 180,E1 22689.475,E2 22689.475} C_VEL
LIN {X 0,Y 506.271,Z 363.874,A -85,B 0,C 180,E1 22686.692,E2 22686.692} C_VEL
LIN {X 0,Y 504.984,Z 362.362,A -85,B 0,C 180,E1 22685.568,E2 22685.568} C_VEL
LIN {X 0,Y 501.08,Z 358.182,A -85,B 0,C 180,E1 22679.886,E2 22679.886} C_VEL
LIN {X 0,Y 500.893,Z 357.811,A -85,B 0,C 180,E1 22677.025,E2 22677.025} C_VEL
LIN {X 0,Y 501.98,Z 359.436,A -85,B 0,C 180,E1 22673.825,E2 22673.825} C_VEL
LIN {X 0,Y 506.03,Z 363.37,A -85,B 0,C 180,E1 22669.296,E2 22669.296} C_VEL
LIN {X 0,Y 510.298,Z 368.521,A -85,B 0,C 180,E1 22666.285,E2 22666.285} C_VEL
LIN {X 0,Y 512.933,Z 371.787,A -85,B 0,C 180,E1 22664.8,E2 22664.8} C_VEL
LIN {X 0,Y 516.477,Z 375.834,A -85,B 0,C 180,E1 22663.06,E2 22663.06} C_VEL
LIN {X 0,Y 521.059,Z 381.345,A -85,B 0,C 180,E1 22661.077,E2 22661.077} C_VEL
LIN {X 0,Y 525.868,Z 387.336,A -85,B 0,C 180,E1 22659.23,E2 22659.23} C_VEL
LIN {X 0,Y 531.135,Z 394.108,A -85,B 0,C 180,E1 22657.416,E2 22657.416} C_VEL
LIN {X 0,Y 538.035,Z 403.165,A -85,B 0,C 180,E1 22655.312,E2 22655.312} C_VEL
LIN {X 0,Y 544.897,Z 412.431,A -85,B 0,C 180,E1 22653.43,E2 22653.43} C_VEL
LIN {X 0,Y 553.827,Z 425.339,A -85,B 0,C 180,E1 22651.21,E2 22651.21} C_VEL
LIN {X 0,Y 563.334,Z 440.027,A -85,B 0,C 180,E1 22649.079,E2 22649.079} C_VEL
LIN {X 0,Y 565.501,Z 444.074,A -85,B 0,C 180,E1 22648.606,E2 22648.606} C_VEL
LIN {X 0,Y 554.794,Z 653.531,A -85,B 0,C 180,E1 22645.36,E2 22645.36} C_VEL
LIN {X 0,Y 546.681,Z 820.654,A -85,B 0,C 180,E1 22642.785,E2 22642.785} C_VEL
LIN {X 0,Y 544.226,Z 848.325,A -85,B 0,C 180,E1 22642.251,E2 22642.251} C_VEL
LIN {X 0,Y 540.965,Z 874.048,A -85,B 0,C 180,E1 22641.577,E2 22641.577} C_VEL
LIN {X 0,Y 537.764,Z 895.448,A -85,B 0,C 180,E1 22640.881,E2 22640.881} C_VEL
LIN {X 0,Y 534.202,Z 916.558,A -85,B 0,C 180,E1 22640.058,E2 22640.058} C_VEL
LIN {X 0,Y 529.602,Z 941.058,A -85,B 0,C 180,E1 22638.926,E2 22638.926} C_VEL
LIN {X 0,Y 524.163,Z 966.551,A -85,B 0,C 180,E1 22637.507,E2 22637.507} C_VEL
LIN {X 0,Y 519.542,Z 986.851,A -85,B 0,C 180,E1 22636.194,E2 22636.194} C_VEL
LIN {X 0,Y 515.009,Z 1005.73,A -85,B 0,C 180,E1 22634.809,E2 22634.809} C_VEL
LIN {X 0,Y 509.897,Z 1026.284,A -85,B 0,C 180,E1 22633.108,E2 22633.108} C_VEL
LIN {X 0,Y 503.839,Z 1049.608,A -85,B 0,C 180,E1 22630.877,E2 22630.877} C_VEL
LIN {X 0,Y 499.248,Z 1067.161,A -85,B 0,C 180,E1 22628.966,E2 22628.966} C_VEL
LIN {X 0,Y 494.94,Z 1083.822,A -85,B 0,C 180,E1 22626.941,E2 22626.941} C_VEL
LIN {X 0,Y 490.015,Z 1103.385,A -85,B 0,C 180,E1 22624.267,E2 22624.267} C_VEL
LIN {X 0,Y 486.048,Z 1119.272,A -85,B 0,C 180,E1 22621.778,E2 22621.778} C_VEL
LIN {X 0,Y 483.021,Z 1132.164,A -85,B 0,C 180,E1 22619.516,E2 22619.516} C_VEL
LIN {X 0,Y 480.343,Z 1144.372,A -85,B 0,C 180,E1 22617.12,E2 22617.12} C_VEL
LIN {X 0,Y 477.886,Z 1156.359,A -85,B 0,C 180,E1 22614.472,E2 22614.472} C_VEL
LIN {X 0,Y 475.595,Z 1169.123,A -85,B 0,C 180,E1 22611.199,E2 22611.199} C_VEL
LIN {X 0,Y 474.171,Z 1178.249,A -85,B 0,C 180,E1 22608.439,E2 22608.439} C_VEL
LIN {X 0,Y 473.255,Z 1185.358,A -85,B 0,C 180,E1 22605.941,E2 22605.941} C_VEL
LIN {X 0,Y 472.691,Z 1190.543,A -85,B 0,C 180,E1 22603.704,E2 22603.704} C_VEL
LIN {X 0,Y 472.249,Z 1195.471,A -85,B 0,C 180,E1 22601.109,E2 22601.109} C_VEL
LIN {X 0,Y 472.048,Z 1199.183,A -85,B 0,C 180,E1 22598.649,E2 22598.649} C_VEL
LIN {X 0,Y 471.95,Z 1201.958,A -85,B 0,C 180,E1 22596.203,E2 22596.203} C_VEL
LIN {X 0,Y 471.915,Z 1203.872,A -85,B 0,C 180,E1 22593.662,E2 22593.662} C_VEL
LIN {X 0,Y 471.913,Z 1204.78,A -85,B 0,C 180,E1 22591.214,E2 22591.214} C_VEL
LIN {X 0,Y 471.913,Z 1204.78,A -85,B 0,C 180,E1 22588.786,E2 22588.786} C_VEL
LIN {X 0,Y 471.915,Z 1203.871,A -85,B 0,C 180,E1 22586.338,E2 22586.338} C_VEL
LIN {X 0,Y 471.949,Z 1201.957,A -85,B 0,C 180,E1 22583.797,E2 22583.797} C_VEL
LIN {X 0,Y 472.056,Z 1199.023,A -85,B 0,C 180,E1 22581.228,E2 22581.228} C_VEL
LIN {X 0,Y 472.296,Z 1194.852,A -85,B 0,C 180,E1 22578.522,E2 22578.522} C_VEL
LIN {X 0,Y 472.952,Z 1188.163,A -85,B 0,C 180,E1 22575.179,E2 22575.179} C_VEL
LIN {X 0,Y 473.854,Z 1180.526,A -85,B 0,C 180,E1 22572.311,E2 22572.311} C_VEL
LIN {X 0,Y 475.088,Z 1172.201,A -85,B 0,C 180,E1 22569.681,E2 22569.681} C_VEL
LIN {X 0,Y 476.66,Z 1163.068,A -85,B 0,C 180,E1 22567.166,E2 22567.166} C_VEL
LIN {X 0,Y 478.662,Z 1152.674,A -85,B 0,C 180,E1 22564.646,E2 22564.646} C_VEL
LIN {X 0,Y 481.716,Z 1138.488,A -85,B 0,C 180,E1 22561.62,E2 22561.62} C_VEL
LIN {X 0,Y 485.209,Z 1123.353,A -85,B 0,C 180,E1 22558.854,E2 22558.854} C_VEL
LIN {X 0,Y 488.591,Z 1109.516,A -85,B 0,C 180,E1 22556.6,E2 22556.6} C_VEL
LIN {X 0,Y 492.26,Z 1095.044,A -85,B 0,C 180,E1 22554.485,E2 22554.485} C_VEL
LIN {X 0,Y 496.567,Z 1078.401,A -85,B 0,C 180,E1 22552.312,E2 22552.312} C_VEL
LIN {X 0,Y 502.179,Z 1056.573,A -85,B 0,C 180,E1 22549.827,E2 22549.827} C_VEL
LIN {X 0,Y 506.747,Z 1038.413,A -85,B 0,C 180,E1 22548.02,E2 22548.02} C_VEL
LIN {X 0,Y 511.034,Z 1020.987,A -85,B 0,C 180,E1 22546.473,E2 22546.473} C_VEL
LIN {X 0,Y 515.368,Z 1002.727,A -85,B 0,C 180,E1 22545.026,E2 22545.026} C_VEL
LIN {X 0,Y 520.681,Z 979.301,A -85,B 0,C 180,E1 22543.393,E2 22543.393} C_VEL
LIN {X 0,Y 525.456,Z 956.027,A -85,B 0,C 180,E1 22542.018,E2 22542.018} C_VEL
LIN {X 0,Y 529.371,Z 935.2,A -85,B 0,C 180,E1 22540.952,E2 22540.952} C_VEL
LIN {X 0,Y 532.91,Z 914.714,A -85,B 0,C 180,E1 22540.049,E2 22540.049} C_VEL
LIN {X 0,Y 536.31,Z 892.649,A -85,B 0,C 180,E1 22539.22,E2 22539.22} C_VEL
LIN {X 0,Y 540.066,Z 863.885,A -85,B 0,C 180,E1 22538.355,E2 22538.355} C_VEL
LIN {X 0,Y 542.505,Z 840.146,A -85,B 0,C 180,E1 22537.812,E2 22537.812} C_VEL
LIN {X 0,Y 544.16,Z 817.718,A -85,B 0,C 180,E1 22537.409,E2 22537.409} C_VEL
LIN {X 0,Y 552.867,Z 605.572,A -85,B 0,C 180,E1 22534.237,E2 22534.237} C_VEL
LIN {X 0,Y 559.774,Z 442.496,A -85,B 0,C 180,E1 22531.769,E2 22531.769} C_VEL
LIN {X 0,Y 543.178,Z 417.599,A -85,B 0,C 180,E1 22528.835,E2 22528.835} C_VEL
LIN {X 0,Y 530.431,Z 399.328,A -85,B 0,C 180,E1 22526.325,E2 22526.325} C_VEL
LIN {X 0,Y 518.949,Z 383.683,A -85,B 0,C 180,E1 22523.837,E2 22523.837} C_VEL
LIN {X 0,Y 507.725,Z 369.177,A -85,B 0,C 180,E1 22521.124,E2 22521.124} C_VEL
LIN {X 0,Y 502.414,Z 362.631,A -85,B 0,C 180,E1 22519.715,E2 22519.715} C_VEL
LIN {X 0,Y 496.751,Z 355.83,A -85,B 0,C 180,E1 22518.119,E2 22518.119} C_VEL
LIN {X 0,Y 493.509,Z 351.993,A -85,B 0,C 180,E1 22517.145,E2 22517.145} C_VEL
LIN {X 0,Y 490.853,Z 348.362,A -85,B 0,C 180,E1 22516.205,E2 22516.205} C_VEL
LIN {X 0,Y 489.408,Z 346.147,A -85,B 0,C 180,E1 22515.403,E2 22515.403} C_VEL
LIN {X 0,Y 487.111,Z 341.881,A -85,B 0,C 180,E1 22513.896,E2 22513.896} C_VEL
LIN {X 0,Y 484.795,Z 338.215,A -85,B 0,C 180,E1 22512.386,E2 22512.386} C_VEL
LIN {X 0,Y 483.856,Z 336.488,A -85,B 0,C 180,E1 22511.684,E2 22511.684} C_VEL
LIN {X 0,Y 481.503,Z 332.731,A -85,B 0,C 180,E1 22509.925,E2 22509.925} C_VEL
LIN {X 0,Y 480.713,Z 331.188,A -85,B 0,C 180,E1 22509.216,E2 22509.216} C_VEL
LIN {X 0,Y 478.169,Z 327.573,A -85,B 0,C 180,E1 22507.087,E2 22507.087} C_VEL
LIN {X 0,Y 477.224,Z 325.626,A -85,B 0,C 180,E1 22506.013,E2 22506.013} C_VEL
LIN {X 0,Y 474.384,Z 321.484,A -85,B 0,C 180,E1 22502.779,E2 22502.779} C_VEL
LIN {X 0,Y 474.121,Z 320.254,A -85,B 0,C 180,E1 22501.571,E2 22501.571} C_VEL
LIN {X 0,Y 474.091,Z 320.153,A -85,B 0,C 180,E1 22497.945,E2 22497.945} C_VEL
LIN {X 0,Y 474.099,Z 320.151,A -85,B 0,C 180,E1 22494.311,E2 22494.311} C_VEL
LIN {X 0,Y 474.111,Z 320.15,A -85,B 0,C 180,E1 22490.74,E2 22490.74} C_VEL
LIN {X 0,Y 474.109,Z 320.15,A -85,B 0,C 180,E1 22487.082,E2 22487.082} C_VEL
LIN {X 0,Y 474.126,Z 320.44,A -85,B 0,C 180,E1 22483.711,E2 22483.711} C_VEL
LIN {X 0,Y 476.491,Z 324.92,A -85,B 0,C 180,E1 22480.254,E2 22480.254} C_VEL
LIN {X 0,Y 477.672,Z 326.342,A -85,B 0,C 180,E1 22479.154,E2 22479.154} C_VEL
LIN {X 0,Y 479.557,Z 330.082,A -85,B 0,C 180,E1 22477.154,E2 22477.154} C_VEL
LIN {X 0,Y 480.983,Z 331.801,A -85,B 0,C 180,E1 22476.085,E2 22476.085} C_VEL
LIN {X 0,Y 482.977,Z 335.617,A -85,B 0,C 180,E1 22474.362,E2 22474.362} C_VEL
LIN {X 0,Y 484.191,Z 337.377,A -85,B 0,C 180,E1 22473.509,E2 22473.509} C_VEL
LIN {X 0,Y 486.539,Z 341.566,A -85,B 0,C 180,E1 22471.792,E2 22471.792} C_VEL
LIN {X 0,Y 489.983,Z 347.545,A -85,B 0,C 180,E1 22469.596,E2 22469.596} C_VEL
LIN {X 0,Y 493.658,Z 352.237,A -85,B 0,C 180,E1 22468.359,E2 22468.359} C_VEL
LIN {X 0,Y 503.489,Z 364.178,A -85,B 0,C 180,E1 22465.563,E2 22465.563} C_VEL
LIN {X 0,Y 509.004,Z 371.228,A -85,B 0,C 180,E1 22464.134,E2 22464.134} C_VEL
LIN {X 0,Y 517.598,Z 382.364,A -85,B 0,C 180,E1 22462.063,E2 22462.063} C_VEL
LIN {X 0,Y 527.895,Z 396.463,A -85,B 0,C 180,E1 22459.803,E2 22459.803} C_VEL
LIN {X 0,Y 538.925,Z 412.267,A -85,B 0,C 180,E1 22457.591,E2 22457.591} C_VEL
LIN {X 0,Y 552.289,Z 432.488,A -85,B 0,C 180,E1 22455.138,E2 22455.138} C_VEL
LIN {X 0,Y 554.625,Z 436.42,A -85,B 0,C 180,E1 22454.727,E2 22454.727} C_VEL
LIN {X 0,Y 544.801,Z 661.792,A -85,B 0,C 180,E1 22451.392,E2 22451.392} C_VEL
LIN {X 0,Y 539.353,Z 788,A -85,B 0,C 180,E1 22449.513,E2 22449.513} C_VEL
LIN {X 0,Y 537.245,Z 814.691,A -85,B 0,C 180,E1 22448.975,E2 22448.975} C_VEL
LIN {X 0,Y 534.578,Z 838.728,A -85,B 0,C 180,E1 22448.309,E2 22448.309} C_VEL
LIN {X 0,Y 531.817,Z 859.463,A -85,B 0,C 180,E1 22447.596,E2 22447.596} C_VEL
LIN {X 0,Y 528.091,Z 883.406,A -85,B 0,C 180,E1 22446.601,E2 22446.601} C_VEL
LIN {X 0,Y 523.725,Z 906.807,A -85,B 0,C 180,E1 22445.41,E2 22445.41} C_VEL
LIN {X 0,Y 520.601,Z 922.243,A -85,B 0,C 180,E1 22444.505,E2 22444.505} C_VEL
LIN {X 0,Y 518.437,Z 929.09,A -85,B 0,C 180,E1 22444.154,E2 22444.154} C_VEL
LIN {X 0,Y 509.727,Z 947.164,A -85,B 0,C 180,E1 22443.399,E2 22443.399} C_VEL
LIN {X 0,Y 507.798,Z 952.629,A -85,B 0,C 180,E1 22443.04,E2 22443.04} C_VEL
LIN {X 0,Y 503.091,Z 971.15,A -85,B 0,C 180,E1 22441.5,E2 22441.5} C_VEL
LIN {X 0,Y 498.253,Z 989.3,A -85,B 0,C 180,E1 22439.779,E2 22439.779} C_VEL
LIN {X 0,Y 492.618,Z 1009.425,A -85,B 0,C 180,E1 22437.566,E2 22437.566} C_VEL
LIN {X 0,Y 488.169,Z 1024.891,A -85,B 0,C 180,E1 22435.605,E2 22435.605} C_VEL
LIN {X 0,Y 483.938,Z 1039.565,A -85,B 0,C 180,E1 22433.5,E2 22433.5} C_VEL
LIN {X 0,Y 479.192,Z 1056.036,A -85,B 0,C 180,E1 22430.776,E2 22430.776} C_VEL
LIN {X 0,Y 475.69,Z 1068.527,A -85,B 0,C 180,E1 22428.378,E2 22428.378} C_VEL
LIN {X 0,Y 472.617,Z 1080.143,A -85,B 0,C 180,E1 22425.837,E2 22425.837} C_VEL
LIN {X 0,Y 469.597,Z 1092.446,A -85,B 0,C 180,E1 22422.668,E2 22422.668} C_VEL
LIN {X 0,Y 467.739,Z 1100.902,A -85,B 0,C 180,E1 22420.095,E2 22420.095} C_VEL
LIN {X 0,Y 466.298,Z 1108.498,A -85,B 0,C 180,E1 22417.392,E2 22417.392} C_VEL
LIN {X 0,Y 465.148,Z 1116.087,A -85,B 0,C 180,E1 22414.068,E2 22414.068} C_VEL
LIN {X 0,Y 464.563,Z 1120.915,A -85,B 0,C 180,E1 22411.357,E2 22411.357} C_VEL
LIN {X 0,Y 464.283,Z 1124.481,A -85,B 0,C 180,E1 22408.766,E2 22408.766} C_VEL
LIN {X 0,Y 464.134,Z 1127.155,A -85,B 0,C 180,E1 22406.047,E2 22406.047} C_VEL
LIN {X 0,Y 464.083,Z 1128.867,A -85,B 0,C 180,E1 22402.821,E2 22402.821} C_VEL
LIN {X 0,Y 464.064,Z 1129.057,A -85,B 0,C 180,E1 22400.075,E2 22400.075} C_VEL
LIN {X 0,Y 464.103,Z 1128.271,A -85,B 0,C 180,E1 22397.559,E2 22397.559} C_VEL
LIN {X 0,Y 464.163,Z 1126.535,A -85,B 0,C 180,E1 22395.019,E2 22395.019} C_VEL
LIN {X 0,Y 464.404,Z 1123.36,A -85,B 0,C 180,E1 22392.069,E2 22392.069} C_VEL
LIN {X 0,Y 464.925,Z 1118.218,A -85,B 0,C 180,E1 22388.82,E2 22388.82} C_VEL
LIN {X 0,Y 465.744,Z 1112.598,A -85,B 0,C 180,E1 22386.062,E2 22386.062} C_VEL
LIN {X 0,Y 467.156,Z 1105.041,A -85,B 0,C 180,E1 22383.016,E2 22383.016} C_VEL
LIN {X 0,Y 469.293,Z 1095.205,A -85,B 0,C 180,E1 22379.814,E2 22379.814} C_VEL
LIN {X 0,Y 471.583,Z 1086.067,A -85,B 0,C 180,E1 22377.272,E2 22377.272} C_VEL
LIN {X 0,Y 474.996,Z 1073.887,A -85,B 0,C 180,E1 22374.332,E2 22374.332} C_VEL
LIN {X 0,Y 479.062,Z 1059.992,A -85,B 0,C 180,E1 22371.508,E2 22371.508} C_VEL
LIN {X 0,Y 483.151,Z 1046.784,A -85,B 0,C 180,E1 22369.16,E2 22369.16} C_VEL
LIN {X 0,Y 488.795,Z 1028.942,A -85,B 0,C 180,E1 22366.421,E2 22366.421} C_VEL
LIN {X 0,Y 493.769,Z 1013.043,A -85,B 0,C 180,E1 22364.318,E2 22364.318} C_VEL
LIN {X 0,Y 498.897,Z 996.52,A -85,B 0,C 180,E1 22362.394,E2 22362.394} C_VEL
LIN {X 0,Y 505.182,Z 975.364,A -85,B 0,C 180,E1 22360.272,E2 22360.272} C_VEL
LIN {X 0,Y 510.376,Z 956.909,A -85,B 0,C 180,E1 22358.68,E2 22358.68} C_VEL
LIN {X 0,Y 515.428,Z 937.9,A -85,B 0,C 180,E1 22357.247,E2 22357.247} C_VEL
LIN {X 0,Y 521.358,Z 913.38,A -85,B 0,C 180,E1 22355.68,E2 22355.68} C_VEL
LIN {X 0,Y 525.786,Z 892.824,A -85,B 0,C 180,E1 22354.572,E2 22354.572} C_VEL
LIN {X 0,Y 529.954,Z 871.232,A -85,B 0,C 180,E1 22353.585,E2 22353.585} C_VEL
LIN {X 0,Y 534.223,Z 844.688,A -85,B 0,C 180,E1 22352.599,E2 22352.599} C_VEL
LIN {X 0,Y 537.104,Z 822.716,A -85,B 0,C 180,E1 22351.954,E2 22351.954} C_VEL
LIN {X 0,Y 539.456,Z 800.336,A -85,B 0,C 180,E1 22351.442,E2 22351.442} C_VEL
LIN {X 0,Y 541.661,Z 766.372,A -85,B 0,C 180,E1 22350.873,E2 22350.873} C_VEL
LIN {X 0,Y 554.08,Z 528.612,A -85,B 0,C 180,E1 22347.28,E2 22347.28} C_VEL
LIN {X 0,Y 558.656,Z 443.979,A -85,B 0,C 180,E1 22345.98,E2 22345.98} C_VEL
LIN {X 0,Y 549.37,Z 429.608,A -85,B 0,C 180,E1 22343.804,E2 22343.804} C_VEL
LIN {X 0,Y 540.733,Z 417.186,A -85,B 0,C 180,E1 22341.563,E2 22341.563} C_VEL
LIN {X 0,Y 532.331,Z 405.692,A -85,B 0,C 180,E1 22339.105,E2 22339.105} C_VEL
LIN {X 0,Y 526.064,Z 397.544,A -85,B 0,C 180,E1 22337.02,E2 22337.02} C_VEL
LIN {X 0,Y 521.683,Z 391.941,A -85,B 0,C 180,E1 22335.394,E2 22335.394} C_VEL
LIN {X 0,Y 517.169,Z 386.299,A -85,B 0,C 180,E1 22333.529,E2 22333.529} C_VEL
LIN {X 0,Y 513.122,Z 381.407,A -85,B 0,C 180,E1 22331.636,E2 22331.636} C_VEL
LIN {X 0,Y 508.892,Z 376.203,A -85,B 0,C 180,E1 22329.272,E2 22329.272} C_VEL
LIN {X 0,Y 505.016,Z 371.557,A -85,B 0,C 180,E1 22326.48,E2 22326.48} C_VEL
LIN {X 0,Y 503.754,Z 370.143,A -85,B 0,C 180,E1 22325.353,E2 22325.353} C_VEL
LIN {X 0,Y 500.064,Z 366.08,A -85,B 0,C 180,E1 22319.771,E2 22319.771} C_VEL
LIN {X 0,Y 499.923,Z 365.777,A -85,B 0,C 180,E1 22316.904,E2 22316.904} C_VEL
LIN {X 0,Y 501.125,Z 367.585,A -85,B 0,C 180,E1 22313.585,E2 22313.585} C_VEL
LIN {X 0,Y 504.912,Z 371.272,A -85,B 0,C 180,E1 22309.387,E2 22309.387} C_VEL
LIN {X 0,Y 509.128,Z 376.406,A -85,B 0,C 180,E1 22306.369,E2 22306.369} C_VEL
LIN {X 0,Y 515.022,Z 383.551,A -85,B 0,C 180,E1 22303.243,E2 22303.243} C_VEL
LIN {X 0,Y 519.419,Z 388.907,A -85,B 0,C 180,E1 22301.306,E2 22301.306} C_VEL
LIN {X 0,Y 524.16,Z 394.915,A -85,B 0,C 180,E1 22299.451,E2 22299.451} C_VEL
LIN {X 0,Y 529.204,Z 401.477,A -85,B 0,C 180,E1 22297.68,E2 22297.68} C_VEL
LIN {X 0,Y 536.25,Z 410.899,A -85,B 0,C 180,E1 22295.491,E2 22295.491} C_VEL
LIN {X 0,Y 542.961,Z 420.14,A -85,B 0,C 180,E1 22293.623,E2 22293.623} C_VEL
LIN {X 0,Y 551.302,Z 432.39,A -85,B 0,C 180,E1 22291.51,E2 22291.51} C_VEL
LIN {X 0,Y 560.367,Z 446.607,A -85,B 0,C 180,E1 22289.433,E2 22289.433} C_VEL
LIN {X 0,Y 561.188,Z 448.34,A -85,B 0,C 180,E1 22289.244,E2 22289.244} C_VEL
LIN {X 0,Y 550.117,Z 657.102,A -85,B 0,C 180,E1 22285.996,E2 22285.996} C_VEL
LIN {X 0,Y 541.893,Z 820.077,A -85,B 0,C 180,E1 22283.47,E2 22283.47} C_VEL
LIN {X 0,Y 539.38,Z 847.691,A -85,B 0,C 180,E1 22282.937,E2 22282.937} C_VEL
LIN {X 0,Y 536,Z 873.525,A -85,B 0,C 180,E1 22282.262,E2 22282.262} C_VEL
LIN {X 0,Y 532.704,Z 894.898,A -85,B 0,C 180,E1 22281.567,E2 22281.567} C_VEL
LIN {X 0,Y 529.164,Z 915.194,A -85,B 0,C 180,E1 22280.778,E2 22280.778} C_VEL
LIN {X 0,Y 524.899,Z 937.09,A -85,B 0,C 180,E1 22279.777,E2 22279.777} C_VEL
LIN {X 0,Y 519.017,Z 964.309,A -85,B 0,C 180,E1 22278.288,E2 22278.288} C_VEL
LIN {X 0,Y 514.012,Z 985.453,A -85,B 0,C 180,E1 22276.922,E2 22276.922} C_VEL
LIN {X 0,Y 509.288,Z 1004.391,A -85,B 0,C 180,E1 22275.532,E2 22275.532} C_VEL
LIN {X 0,Y 504.653,Z 1022.197,A -85,B 0,C 180,E1 22274.061,E2 22274.061} C_VEL
LIN {X 0,Y 498.854,Z 1044.053,A -85,B 0,C 180,E1 22272.024,E2 22272.024} C_VEL
LIN {X 0,Y 492.943,Z 1065.36,A -85,B 0,C 180,E1 22269.712,E2 22269.712} C_VEL
LIN {X 0,Y 488.384,Z 1082.052,A -85,B 0,C 180,E1 22267.67,E2 22267.67} C_VEL
LIN {X 0,Y 483.85,Z 1098.994,A -85,B 0,C 180,E1 22265.353,E2 22265.353} C_VEL
LIN {X 0,Y 479.018,Z 1117.644,A -85,B 0,C 180,E1 22262.442,E2 22262.442} C_VEL
LIN {X 0,Y 475.553,Z 1131.56,A -85,B 0,C 180,E1 22259.972,E2 22259.972} C_VEL
LIN {X 0,Y 472.797,Z 1143.534,A -85,B 0,C 180,E1 22257.59,E2 22257.59} C_VEL
LIN {X 0,Y 470.33,Z 1155.002,A -85,B 0,C 180,E1 22255.027,E2 22255.027} C_VEL
LIN {X 0,Y 467.945,Z 1167.488,A -85,B 0,C 180,E1 22251.826,E2 22251.826} C_VEL
LIN {X 0,Y 466.313,Z 1177.507,A -85,B 0,C 180,E1 22248.761,E2 22248.761} C_VEL
LIN {X 0,Y 465.307,Z 1184.826,A -85,B 0,C 180,E1 22246.146,E2 22246.146} C_VEL
LIN {X 0,Y 464.686,Z 1190.665,A -85,B 0,C 180,E1 22243.691,E2 22243.691} C_VEL
LIN {X 0,Y 464.26,Z 1195.627,A -85,B 0,C 180,E1 22241.176,E2 22241.176} C_VEL
LIN {X 0,Y 464.059,Z 1199.181,A -85,B 0,C 180,E1 22238.8,E2 22238.8} C_VEL
LIN {X 0,Y 463.954,Z 1201.955,A -85,B 0,C 180,E1 22236.31,E2 22236.31} C_VEL
LIN {X 0,Y 463.914,Z 1203.811,A -85,B 0,C 180,E1 22233.831,E2 22233.831} C_VEL
LIN {X 0,Y 463.913,Z 1204.757,A -85,B 0,C 180,E1 22231.359,E2 22231.359} C_VEL
LIN {X 0,Y 463.911,Z 1204.802,A -85,B 0,C 180,E1 22228.889,E2 22228.889} C_VEL
LIN {X 0,Y 463.914,Z 1203.947,A -85,B 0,C 180,E1 22226.417,E2 22226.417} C_VEL
LIN {X 0,Y 463.947,Z 1202.181,A -85,B 0,C 180,E1 22223.938,E2 22223.938} C_VEL
LIN {X 0,Y 464.044,Z 1199.499,A -85,B 0,C 180,E1 22221.45,E2 22221.45} C_VEL
LIN {X 0,Y 464.235,Z 1196.06,A -85,B 0,C 180,E1 22219.075,E2 22219.075} C_VEL
LIN {X 0,Y 464.631,Z 1191.22,A -85,B 0,C 180,E1 22216.561,E2 22216.561} C_VEL
LIN {X 0,Y 465.257,Z 1185.314,A -85,B 0,C 180,E1 22214.033,E2 22214.033} C_VEL
LIN {X 0,Y 466.22,Z 1178.142,A -85,B 0,C 180,E1 22211.433,E2 22211.433} C_VEL
LIN {X 0,Y 467.575,Z 1169.741,A -85,B 0,C 180,E1 22208.808,E2 22208.808} C_VEL
LIN {X 0,Y 469.811,Z 1157.923,A -85,B 0,C 180,E1 22205.615,E2 22205.615} C_VEL
LIN {X 0,Y 472.556,Z 1145.026,A -85,B 0,C 180,E1 22202.669,E2 22202.669} C_VEL
LIN {X 0,Y 475.332,Z 1133.006,A -85,B 0,C 180,E1 22200.236,E2 22200.236} C_VEL
LIN {X 0,Y 478.47,Z 1120.323,A -85,B 0,C 180,E1 22197.942,E2 22197.942} C_VEL
LIN {X 0,Y 482.366,Z 1105.427,A -85,B 0,C 180,E1 22195.537,E2 22195.537} C_VEL
LIN {X 0,Y 487.687,Z 1085.311,A -85,B 0,C 180,E1 22192.703,E2 22192.703} C_VEL
LIN {X 0,Y 492.19,Z 1068.367,A -85,B 0,C 180,E1 22190.62,E2 22190.62} C_VEL
LIN {X 0,Y 496.545,Z 1051.948,A -85,B 0,C 180,E1 22188.818,E2 22188.818} C_VEL
LIN {X 0,Y 501.393,Z 1033.368,A -85,B 0,C 180,E1 22187,E2 22187} C_VEL
LIN {X 0,Y 507.559,Z 1008.771,A -85,B 0,C 180,E1 22184.912,E2 22184.912} C_VEL
LIN {X 0,Y 512.287,Z 988.761,A -85,B 0,C 180,E1 22183.444,E2 22183.444} C_VEL
LIN {X 0,Y 516.678,Z 969.018,A -85,B 0,C 180,E1 22182.169,E2 22182.169} C_VEL
LIN {X 0,Y 521.316,Z 946.729,A -85,B 0,C 180,E1 22180.916,E2 22180.916} C_VEL
LIN {X 0,Y 526.355,Z 919.504,A -85,B 0,C 180,E1 22179.633,E2 22179.633} C_VEL
LIN {X 0,Y 529.94,Z 897.424,A -85,B 0,C 180,E1 22178.772,E2 22178.772} C_VEL
LIN {X 0,Y 533.02,Z 875.837,A -85,B 0,C 180,E1 22178.07,E2 22178.07} C_VEL
LIN {X 0,Y 535.797,Z 852.801,A -85,B 0,C 180,E1 22177.459,E2 22177.459} C_VEL
LIN {X 0,Y 538.482,Z 822.764,A -85,B 0,C 180,E1 22176.863,E2 22176.863} C_VEL
LIN {X 0,Y 541.61,Z 752.122,A -85,B 0,C 180,E1 22175.787,E2 22175.787} C_VEL
LIN {X 0,Y 551.056,Z 531.196,A -85,B 0,C 180,E1 22172.466,E2 22172.466} C_VEL
LIN {X 0,Y 554.687,Z 446.475,A -85,B 0,C 180,E1 22171.155,E2 22171.155} C_VEL
LIN {X 0,Y 539.186,Z 423.052,A -85,B 0,C 180,E1 22168.342,E2 22168.342} C_VEL
LIN {X 0,Y 527.189,Z 405.686,A -85,B 0,C 180,E1 22165.924,E2 22165.924} C_VEL
LIN {X 0,Y 515.953,Z 390.235,A -85,B 0,C 180,E1 22163.439,E2 22163.439} C_VEL
LIN {X 0,Y 505.195,Z 376.164,A -85,B 0,C 180,E1 22160.78,E2 22160.78} C_VEL
LIN {X 0,Y 500.041,Z 369.731,A -85,B 0,C 180,E1 22159.386,E2 22159.386} C_VEL
LIN {X 0,Y 492.33,Z 360.213,A -85,B 0,C 180,E1 22157.127,E2 22157.127} C_VEL
LIN {X 0,Y 487.215,Z 354.142,A -85,B 0,C 180,E1 22155.474,E2 22155.474} C_VEL
LIN {X 0,Y 483.482,Z 349.608,A -85,B 0,C 180,E1 22154.156,E2 22154.156} C_VEL
LIN {X 0,Y 482.222,Z 347.987,A -85,B 0,C 180,E1 22153.551,E2 22153.551} C_VEL
LIN {X 0,Y 480.1,Z 344.102,A -85,B 0,C 180,E1 22152.021,E2 22152.021} C_VEL
LIN {X 0,Y 476.987,Z 338.984,A -85,B 0,C 180,E1 22149.654,E2 22149.654} C_VEL
LIN {X 0,Y 475.953,Z 337.429,A -85,B 0,C 180,E1 22148.822,E2 22148.822} C_VEL
LIN {X 0,Y 473.644,Z 333.623,A -85,B 0,C 180,E1 22146.668,E2 22146.668} C_VEL
LIN {X 0,Y 472.706,Z 332.134,A -85,B 0,C 180,E1 22145.706,E2 22145.706} C_VEL
LIN {X 0,Y 469.997,Z 327.723,A -85,B 0,C 180,E1 22142.317,E2 22142.317} C_VEL
LIN {X 0,Y 468.945,Z 326.275,A -85,B 0,C 180,E1 22140.733,E2 22140.733} C_VEL
LIN {X 0,Y 466.772,Z 323.356,A -85,B 0,C 180,E1 22135.331,E2 22135.331} C_VEL
LIN {X 0,Y 466.606,Z 323.002,A -85,B 0,C 180,E1 22131.993,E2 22131.993} C_VEL
LIN {X 0,Y 467.195,Z 324.204,A -85,B 0,C 180,E1 22128.394,E2 22128.394} C_VEL
LIN {X 0,Y 469.78,Z 327.231,A -85,B 0,C 180,E1 22123.683,E2 22123.683} C_VEL
LIN {X 0,Y 472.161,Z 331.627,A -85,B 0,C 180,E1 22120.323,E2 22120.323} C_VEL
LIN {X 0,Y 473.31,Z 333.087,A -85,B 0,C 180,E1 22119.212,E2 22119.212} C_VEL
LIN {X 0,Y 475.289,Z 336.876,A -85,B 0,C 180,E1 22117.133,E2 22117.133} C_VEL
LIN {X 0,Y 476.569,Z 338.61,A -85,B 0,C 180,E1 22116.113,E2 22116.113} C_VEL
LIN {X 0,Y 478.756,Z 342.531,A -85,B 0,C 180,E1 22114.252,E2 22114.252} C_VEL
LIN {X 0,Y 479.695,Z 344.208,A -85,B 0,C 180,E1 22113.508,E2 22113.508} C_VEL
LIN {X 0,Y 482.109,Z 348.157,A -85,B 0,C 180,E1 22111.914,E2 22111.914} C_VEL
LIN {X 0,Y 486.826,Z 353.835,A -85,B 0,C 180,E1 22110.195,E2 22110.195} C_VEL
LIN {X 0,Y 493.925,Z 362.5,A -85,B 0,C 180,E1 22107.934,E2 22107.934} C_VEL
LIN {X 0,Y 501.776,Z 372.234,A -85,B 0,C 180,E1 22105.706,E2 22105.706} C_VEL
LIN {X 0,Y 506.749,Z 378.565,A -85,B 0,C 180,E1 22104.403,E2 22104.403} C_VEL
LIN {X 0,Y 515.815,Z 390.452,A -85,B 0,C 180,E1 22102.19,E2 22102.19} C_VEL
LIN {X 0,Y 527.709,Z 407.043,A -85,B 0,C 180,E1 22099.572,E2 22099.572} C_VEL
LIN {X 0,Y 540.086,Z 425.282,A -85,B 0,C 180,E1 22097.109,E2 22097.109} C_VEL
LIN {X 0,Y 549.687,Z 440.449,A -85,B 0,C 180,E1 22095.339,E2 22095.339} C_VEL
LIN {X 0,Y 539.537,Z 665.526,A -85,B 0,C 180,E1 22091.992,E2 22091.992} C_VEL
LIN {X 0,Y 534.059,Z 788.255,A -85,B 0,C 180,E1 22090.154,E2 22090.154} C_VEL
LIN {X 0,Y 531.908,Z 814.88,A -85,B 0,C 180,E1 22089.617,E2 22089.617} C_VEL
LIN {X 0,Y 529.149,Z 839.061,A -85,B 0,C 180,E1 22088.945,E2 22088.945} C_VEL
LIN {X 0,Y 526.319,Z 859.742,A -85,B 0,C 180,E1 22088.231,E2 22088.231} C_VEL
LIN {X 0,Y 522.552,Z 883.363,A -85,B 0,C 180,E1 22087.249,E2 22087.249} C_VEL
LIN {X 0,Y 518.082,Z 906.73,A -85,B 0,C 180,E1 22086.059,E2 22086.059} C_VEL
LIN {X 0,Y 514.121,Z 925.536,A -85,B 0,C 180,E1 22084.941,E2 22084.941} C_VEL
LIN {X 0,Y 509.783,Z 944.53,A -85,B 0,C 180,E1 22083.647,E2 22083.647} C_VEL
LIN {X 0,Y 507.798,Z 952.629,A -85,B 0,C 180,E1 22083.04,E2 22083.04} C_VEL
LIN {X 0,Y 505.44,Z 959.052,A -85,B 0,C 180,E1 22082.612,E2 22082.612} C_VEL
LIN {X 0,Y 496.726,Z 975.301,A -85,B 0,C 180,E1 22081.703,E2 22081.703} C_VEL
LIN {X 0,Y 494.306,Z 981.31,A -85,B 0,C 180,E1 22081.212,E2 22081.212} C_VEL
LIN {X 0,Y 489.371,Z 998.625,A -85,B 0,C 180,E1 22079.431,E2 22079.431} C_VEL
LIN {X 0,Y 484.874,Z 1013.962,A -85,B 0,C 180,E1 22077.644,E2 22077.644} C_VEL
LIN {X 0,Y 479.624,Z 1031.666,A -85,B 0,C 180,E1 22075.3,E2 22075.3} C_VEL
LIN {X 0,Y 474.713,Z 1047.74,A -85,B 0,C 180,E1 22072.802,E2 22072.802} C_VEL
LIN {X 0,Y 470.866,Z 1060.682,A -85,B 0,C 180,E1 22070.51,E2 22070.51} C_VEL
LIN {X 0,Y 466.921,Z 1074.512,A -85,B 0,C 180,E1 22067.703,E2 22067.703} C_VEL
LIN {X 0,Y 463.695,Z 1086.314,A -85,B 0,C 180,E1 22064.868,E2 22064.868} C_VEL
LIN {X 0,Y 461.352,Z 1095.724,A -85,B 0,C 180,E1 22062.262,E2 22062.262} C_VEL
LIN {X 0,Y 459.192,Z 1105.632,A -85,B 0,C 180,E1 22059.02,E2 22059.02} C_VEL
LIN {X 0,Y 457.864,Z 1112.787,A -85,B 0,C 180,E1 22056.143,E2 22056.143} C_VEL
LIN {X 0,Y 457.031,Z 1118.438,A -85,B 0,C 180,E1 22053.386,E2 22053.386} C_VEL
LIN {X 0,Y 456.478,Z 1123.529,A -85,B 0,C 180,E1 22050.251,E2 22050.251} C_VEL
LIN {X 0,Y 456.203,Z 1126.98,A -85,B 0,C 180,E1 22047.11,E2 22047.11} C_VEL
LIN {X 0,Y 456.114,Z 1128.838,A -85,B 0,C 180,E1 22044.465,E2 22044.465} C_VEL
LIN {X 0,Y 456.108,Z 1129.704,A -85,B 0,C 180,E1 22041.808,E2 22041.808} C_VEL
LIN {X 0,Y 456.114,Z 1129.491,A -85,B 0,C 180,E1 22038.621,E2 22038.621} C_VEL
LIN {X 0,Y 456.195,Z 1127.719,A -85,B 0,C 180,E1 22035.531,E2 22035.531} C_VEL
LIN {X 0,Y 456.362,Z 1125.225,A -85,B 0,C 180,E1 22032.927,E2 22032.927} C_VEL
LIN {X 0,Y 456.698,Z 1121.719,A -85,B 0,C 180,E1 22030.295,E2 22030.295} C_VEL
LIN {X 0,Y 457.477,Z 1116.185,A -85,B 0,C 180,E1 22027.105,E2 22027.105} C_VEL
LIN {X 0,Y 458.769,Z 1108.826,A -85,B 0,C 180,E1 22023.88,E2 22023.88} C_VEL
LIN {X 0,Y 460.391,Z 1101.42,A -85,B 0,C 180,E1 22021.175,E2 22021.175} C_VEL
LIN {X 0,Y 462.96,Z 1091.374,A -85,B 0,C 180,E1 22018.053,E2 22018.053} C_VEL
LIN {X 0,Y 466.263,Z 1079.517,A -85,B 0,C 180,E1 22015.004,E2 22015.004} C_VEL
LIN {X 0,Y 469.693,Z 1068.297,A -85,B 0,C 180,E1 22012.496,E2 22012.496} C_VEL
LIN {X 0,Y 474.682,Z 1052.768,A -85,B 0,C 180,E1 22009.502,E2 22009.502} C_VEL
LIN {X 0,Y 479.326,Z 1038.557,A -85,B 0,C 180,E1 22007.154,E2 22007.154} C_VEL
LIN {X 0,Y 484.249,Z 1023.703,A -85,B 0,C 180,E1 22004.994,E2 22004.994} C_VEL
LIN {X 0,Y 490.498,Z 1004.616,A -85,B 0,C 180,E1 22002.593,E2 22002.593} C_VEL
LIN {X 0,Y 495.648,Z 988.276,A -85,B 0,C 180,E1 22000.815,E2 22000.815} C_VEL
LIN {X 0,Y 500.721,Z 971.607,A -85,B 0,C 180,E1 21999.216,E2 21999.216} C_VEL
LIN {X 0,Y 506.664,Z 951.191,A -85,B 0,C 180,E1 21997.504,E2 21997.504} C_VEL
LIN {X 0,Y 512.478,Z 929.084,A -85,B 0,C 180,E1 21995.936,E2 21995.936} C_VEL
LIN {X 0,Y 516.87,Z 910.963,A -85,B 0,C 180,E1 21994.826,E2 21994.826} C_VEL
LIN {X 0,Y 521.064,Z 891.913,A -85,B 0,C 180,E1 21993.811,E2 21993.811} C_VEL
LIN {X 0,Y 525.891,Z 867.403,A -85,B 0,C 180,E1 21992.711,E2 21992.711} C_VEL
LIN {X 0,Y 529.736,Z 843.319,A -85,B 0,C 180,E1 21991.845,E2 21991.845} C_VEL
LIN {X 0,Y 532.625,Z 821.574,A -85,B 0,C 180,E1 21991.215,E2 21991.215} C_VEL
LIN {X 0,Y 535.346,Z 795.496,A -85,B 0,C 180,E1 21990.638,E2 21990.638} C_VEL
LIN {X 0,Y 537.991,Z 750.191,A -85,B 0,C 180,E1 21989.922,E2 21989.922} C_VEL
LIN {X 0,Y 551.018,Z 511.001,A -85,B 0,C 180,E1 21986.294,E2 21986.294} C_VEL
LIN {X 0,Y 554.524,Z 448.474,A -85,B 0,C 180,E1 21985.328,E2 21985.328} C_VEL
LIN {X 0,Y 545.548,Z 434.65,A -85,B 0,C 180,E1 21983.15,E2 21983.15} C_VEL
LIN {X 0,Y 538.021,Z 423.728,A -85,B 0,C 180,E1 21981.134,E2 21981.134} C_VEL
LIN {X 0,Y 530.044,Z 412.596,A -85,B 0,C 180,E1 21978.733,E2 21978.733} C_VEL
LIN {X 0,Y 524.04,Z 404.736,A -85,B 0,C 180,E1 21976.688,E2 21976.688} C_VEL
LIN {X 0,Y 519.877,Z 399.325,A -85,B 0,C 180,E1 21975.106,E2 21975.106} C_VEL
LIN {X 0,Y 515.569,Z 393.835,A -85,B 0,C 180,E1 21973.286,E2 21973.286} C_VEL
LIN {X 0,Y 511.703,Z 389.091,A -85,B 0,C 180,E1 21971.44,E2 21971.44} C_VEL
LIN {X 0,Y 507.552,Z 383.927,A -85,B 0,C 180,E1 21969.068,E2 21969.068} C_VEL
LIN {X 0,Y 503.645,Z 379.032,A -85,B 0,C 180,E1 21966.154,E2 21966.154} C_VEL
LIN {X 0,Y 499.519,Z 374.736,A -85,B 0,C 180,E1 21961.032,E2 21961.032} C_VEL
LIN {X 0,Y 498.851,Z 373.607,A -85,B 0,C 180,E1 21958.047,E2 21958.047} C_VEL
LIN {X 0,Y 499.378,Z 374.438,A -85,B 0,C 180,E1 21955.176,E2 21955.176} C_VEL
LIN {X 0,Y 503.672,Z 378.979,A -85,B 0,C 180,E1 21949.592,E2 21949.592} C_VEL
LIN {X 0,Y 507.966,Z 384.292,A -85,B 0,C 180,E1 21946.453,E2 21946.453} C_VEL
LIN {X 0,Y 513.463,Z 391.099,A -85,B 0,C 180,E1 21943.482,E2 21943.482} C_VEL
LIN {X 0,Y 517.787,Z 396.468,A -85,B 0,C 180,E1 21941.537,E2 21941.537} C_VEL
LIN {X 0,Y 522.521,Z 402.582,A -85,B 0,C 180,E1 21939.65,E2 21939.65} C_VEL
LIN {X 0,Y 527.287,Z 408.846,A -85,B 0,C 180,E1 21937.947,E2 21937.947} C_VEL
LIN {X 0,Y 534.229,Z 418.29,A -85,B 0,C 180,E1 21935.743,E2 21935.743} C_VEL
LIN {X 0,Y 541.308,Z 428.238,A -85,B 0,C 180,E1 21933.743,E2 21933.743} C_VEL
LIN {X 0,Y 548.994,Z 439.752,A -85,B 0,C 180,E1 21931.765,E2 21931.765} C_VEL
LIN {X 0,Y 556.951,Z 452.413,A -85,B 0,C 180,E1 21929.897,E2 21929.897} C_VEL
LIN {X 0,Y 545.648,Z 658.313,A -85,B 0,C 180,E1 21926.68,E2 21926.68} C_VEL
LIN {X 0,Y 537.178,Z 819.853,A -85,B 0,C 180,E1 21924.163,E2 21924.163} C_VEL
LIN {X 0,Y 534.56,Z 847.634,A -85,B 0,C 180,E1 21923.624,E2 21923.624} C_VEL
LIN {X 0,Y 531.119,Z 873.097,A -85,B 0,C 180,E1 21922.959,E2 21922.959} C_VEL
LIN {X 0,Y 527.731,Z 894.379,A -85,B 0,C 180,E1 21922.266,E2 21922.266} C_VEL
LIN {X 0,Y 524.036,Z 914.839,A -85,B 0,C 180,E1 21921.47,E2 21921.47} C_VEL
LIN {X 0,Y 519.71,Z 936.336,A -85,B 0,C 180,E1 21920.486,E2 21920.486} C_VEL
LIN {X 0,Y 513.655,Z 963.411,A -85,B 0,C 180,E1 21919.003,E2 21919.003} C_VEL
LIN {X 0,Y 508.572,Z 984.128,A -85,B 0,C 180,E1 21917.665,E2 21917.665} C_VEL
LIN {X 0,Y 503.798,Z 1002.524,A -85,B 0,C 180,E1 21916.316,E2 21916.316} C_VEL
LIN {X 0,Y 498.815,Z 1020.904,A -85,B 0,C 180,E1 21914.797,E2 21914.797} C_VEL
LIN {X 0,Y 493.092,Z 1041.538,A -85,B 0,C 180,E1 21912.867,E2 21912.867} C_VEL
LIN {X 0,Y 486.749,Z 1063.633,A -85,B 0,C 180,E1 21910.475,E2 21910.475} C_VEL
LIN {X 0,Y 481.94,Z 1080.358,A -85,B 0,C 180,E1 21908.415,E2 21908.415} C_VEL
LIN {X 0,Y 477.54,Z 1095.899,A -85,B 0,C 180,E1 21906.28,E2 21906.28} C_VEL
LIN {X 0,Y 472.654,Z 1113.848,A -85,B 0,C 180,E1 21903.513,E2 21903.513} C_VEL
LIN {X 0,Y 468.42,Z 1129.854,A -85,B 0,C 180,E1 21900.655,E2 21900.655} C_VEL
LIN {X 0,Y 465.411,Z 1142.081,A -85,B 0,C 180,E1 21898.205,E2 21898.205} C_VEL
LIN {X 0,Y 462.934,Z 1153.089,A -85,B 0,C 180,E1 21895.73,E2 21895.73} C_VEL
LIN {X 0,Y 460.727,Z 1163.853,A -85,B 0,C 180,E1 21892.994,E2 21892.994} C_VEL
LIN {X 0,Y 458.641,Z 1175.624,A -85,B 0,C 180,E1 21889.484,E2 21889.484} C_VEL
LIN {X 0,Y 457.46,Z 1183.583,A -85,B 0,C 180,E1 21886.638,E2 21886.638} C_VEL
LIN {X 0,Y 456.77,Z 1189.682,A -85,B 0,C 180,E1 21884.062,E2 21884.062} C_VEL
LIN {X 0,Y 456.29,Z 1194.94,A -85,B 0,C 180,E1 21881.374,E2 21881.374} C_VEL
LIN {X 0,Y 456.065,Z 1198.893,A -85,B 0,C 180,E1 21878.828,E2 21878.828} C_VEL
LIN {X 0,Y 455.955,Z 1201.837,A -85,B 0,C 180,E1 21876.295,E2 21876.295} C_VEL
LIN {X 0,Y 455.914,Z 1203.717,A -85,B 0,C 180,E1 21873.898,E2 21873.898} C_VEL
LIN {X 0,Y 455.91,Z 1204.703,A -85,B 0,C 180,E1 21871.508,E2 21871.508} C_VEL
LIN {X 0,Y 455.908,Z 1204.798,A -85,B 0,C 180,E1 21868.995,E2 21868.995} C_VEL
LIN {X 0,Y 455.915,Z 1203.936,A -85,B 0,C 180,E1 21866.48,E2 21866.48} C_VEL
LIN {X 0,Y 455.948,Z 1202.083,A -85,B 0,C 180,E1 21863.958,E2 21863.958} C_VEL
LIN {X 0,Y 456.048,Z 1199.244,A -85,B 0,C 180,E1 21861.426,E2 21861.426} C_VEL
LIN {X 0,Y 456.26,Z 1195.403,A -85,B 0,C 180,E1 21858.881,E2 21858.881} C_VEL
LIN {X 0,Y 456.711,Z 1190.268,A -85,B 0,C 180,E1 21856.194,E2 21856.194} C_VEL
LIN {X 0,Y 457.371,Z 1184.298,A -85,B 0,C 180,E1 21853.62,E2 21853.62} C_VEL
LIN {X 0,Y 458.398,Z 1177.241,A -85,B 0,C 180,E1 21851.035,E2 21851.035} C_VEL
LIN {X 0,Y 459.935,Z 1168.158,A -85,B 0,C 180,E1 21848.17,E2 21848.17} C_VEL
LIN {X 0,Y 462.593,Z 1154.994,A -85,B 0,C 180,E1 21844.662,E2 21844.662} C_VEL
LIN {X 0,Y 465.161,Z 1143.646,A -85,B 0,C 180,E1 21842.057,E2 21842.057} C_VEL
LIN {X 0,Y 468.128,Z 1131.543,A -85,B 0,C 180,E1 21839.589,E2 21839.589} C_VEL
LIN {X 0,Y 471.475,Z 1118.756,A -85,B 0,C 180,E1 21837.263,E2 21837.263} C_VEL
LIN {X 0,Y 476.018,Z 1102.083,A -85,B 0,C 180,E1 21834.569,E2 21834.569} C_VEL
LIN {X 0,Y 481.123,Z 1083.409,A -85,B 0,C 180,E1 21831.967,E2 21831.967} C_VEL
LIN {X 0,Y 485.523,Z 1067.525,A -85,B 0,C 180,E1 21830.005,E2 21830.005} C_VEL
LIN {X 0,Y 490.125,Z 1050.791,A -85,B 0,C 180,E1 21828.158,E2 21828.158} C_VEL
LIN {X 0,Y 495.521,Z 1030.838,A -85,B 0,C 180,E1 21826.203,E2 21826.203} C_VEL
LIN {X 0,Y 501.574,Z 1007.37,A -85,B 0,C 180,E1 21824.222,E2 21824.222} C_VEL
LIN {X 0,Y 506.3,Z 987.953,A -85,B 0,C 180,E1 21822.794,E2 21822.794} C_VEL
LIN {X 0,Y 510.79,Z 968.378,A -85,B 0,C 180,E1 21821.524,E2 21821.524} C_VEL
LIN {X 0,Y 515.357,Z 947.041,A -85,B 0,C 180,E1 21820.318,E2 21820.318} C_VEL
LIN {X 0,Y 520.608,Z 919.64,A -85,B 0,C 180,E1 21819.015,E2 21819.015} C_VEL
LIN {X 0,Y 524.362,Z 897.219,A -85,B 0,C 180,E1 21818.135,E2 21818.135} C_VEL
LIN {X 0,Y 527.516,Z 875.801,A -85,B 0,C 180,E1 21817.436,E2 21817.436} C_VEL
LIN {X 0,Y 530.308,Z 853.299,A -85,B 0,C 180,E1 21816.835,E2 21816.835} C_VEL
LIN {X 0,Y 533.085,Z 823.639,A -85,B 0,C 180,E1 21816.237,E2 21816.237} C_VEL
LIN {X 0,Y 535.882,Z 763.806,A -85,B 0,C 180,E1 21815.316,E2 21815.316} C_VEL
LIN {X 0,Y 545.659,Z 542.255,A -85,B 0,C 180,E1 21811.968,E2 21811.968} C_VEL
LIN {X 0,Y 549.78,Z 450.574,A -85,B 0,C 180,E1 21810.553,E2 21810.553} C_VEL
LIN {X 0,Y 533.817,Z 426.293,A -85,B 0,C 180,E1 21807.559,E2 21807.559} C_VEL
LIN {X 0,Y 521.39,Z 408.318,A -85,B 0,C 180,E1 21804.955,E2 21804.955} C_VEL
LIN {X 0,Y 510.565,Z 393.513,A -85,B 0,C 180,E1 21802.451,E2 21802.451} C_VEL
LIN {X 0,Y 501.992,Z 382.338,A -85,B 0,C 180,E1 21800.248,E2 21800.248} C_VEL
LIN {X 0,Y 497.779,Z 376.934,A -85,B 0,C 180,E1 21799.082,E2 21799.082} C_VEL
LIN {X 0,Y 490.079,Z 367.363,A -85,B 0,C 180,E1 21796.78,E2 21796.78} C_VEL
LIN {X 0,Y 485.212,Z 361.493,A -85,B 0,C 180,E1 21795.172,E2 21795.172} C_VEL
LIN {X 0,Y 481.386,Z 356.687,A -85,B 0,C 180,E1 21793.789,E2 21793.789} C_VEL
LIN {X 0,Y 476.909,Z 351.865,A -85,B 0,C 180,E1 21792.072,E2 21792.072} C_VEL
LIN {X 0,Y 475.181,Z 349.727,A -85,B 0,C 180,E1 21791.347,E2 21791.347} C_VEL
LIN {X 0,Y 472.9,Z 346.444,A -85,B 0,C 180,E1 21789.861,E2 21789.861} C_VEL
LIN {X 0,Y 472.037,Z 344.555,A -85,B 0,C 180,E1 21789.018,E2 21789.018} C_VEL
LIN {X 0,Y 469.475,Z 340.678,A -85,B 0,C 180,E1 21786.727,E2 21786.727} C_VEL
LIN {X 0,Y 468.762,Z 339.17,A -85,B 0,C 180,E1 21785.877,E2 21785.877} C_VEL
LIN {X 0,Y 465.922,Z 334.835,A -85,B 0,C 180,E1 21782.46,E2 21782.46} C_VEL
LIN {X 0,Y 465.093,Z 333.388,A -85,B 0,C 180,E1 21781.109,E2 21781.109} C_VEL
LIN {X 0,Y 462.667,Z 330.295,A -85,B 0,C 180,E1 21775.538,E2 21775.538} C_VEL
LIN {X 0,Y 462.476,Z 329.833,A -85,B 0,C 180,E1 21772.171,E2 21772.171} C_VEL
LIN {X 0,Y 463.01,Z 330.976,A -85,B 0,C 180,E1 21768.54,E2 21768.54} C_VEL
LIN {X 0,Y 465.517,Z 333.984,A -85,B 0,C 180,E1 21763.757,E2 21763.757} C_VEL
LIN {X 0,Y 467.966,Z 338.469,A -85,B 0,C 180,E1 21760.27,E2 21760.27} C_VEL
LIN {X 0,Y 468.951,Z 339.828,A -85,B 0,C 180,E1 21759.271,E2 21759.271} C_VEL
LIN {X 0,Y 470.822,Z 343.458,A -85,B 0,C 180,E1 21757.262,E2 21757.262} C_VEL
LIN {X 0,Y 472.045,Z 345.086,A -85,B 0,C 180,E1 21756.268,E2 21756.268} C_VEL
LIN {X 0,Y 474.01,Z 348.63,A -85,B 0,C 180,E1 21754.712,E2 21754.712} C_VEL
LIN {X 0,Y 476.237,Z 351.164,A -85,B 0,C 180,E1 21753.737,E2 21753.737} C_VEL
LIN {X 0,Y 481.41,Z 357.181,A -85,B 0,C 180,E1 21751.717,E2 21751.717} C_VEL
LIN {X 0,Y 486.494,Z 363.221,A -85,B 0,C 180,E1 21749.935,E2 21749.935} C_VEL
LIN {X 0,Y 492.556,Z 370.716,A -85,B 0,C 180,E1 21748.006,E2 21748.006} C_VEL
LIN {X 0,Y 499.581,Z 379.567,A -85,B 0,C 180,E1 21745.985,E2 21745.985} C_VEL
LIN {X 0,Y 504.502,Z 385.899,A -85,B 0,C 180,E1 21744.674,E2 21744.674} C_VEL
LIN {X 0,Y 513.752,Z 398.256,A -85,B 0,C 180,E1 21742.382,E2 21742.382} C_VEL
LIN {X 0,Y 525.032,Z 414.166,A -85,B 0,C 180,E1 21739.86,E2 21739.86} C_VEL
LIN {X 0,Y 537.358,Z 432.632,A -85,B 0,C 180,E1 21737.366,E2 21737.366} C_VEL
LIN {X 0,Y 544.811,Z 444.482,A -85,B 0,C 180,E1 21735.961,E2 21735.961} C_VEL
LIN {X 0,Y 534.279,Z 670.392,A -85,B 0,C 180,E1 21732.586,E2 21732.586} C_VEL
LIN {X 0,Y 528.804,Z 788.818,A -85,B 0,C 180,E1 21730.802,E2 21730.802} C_VEL
LIN {X 0,Y 526.562,Z 815.653,A -85,B 0,C 180,E1 21730.256,E2 21730.256} C_VEL
LIN {X 0,Y 523.759,Z 839.6,A -85,B 0,C 180,E1 21729.587,E2 21729.587} C_VEL
LIN {X 0,Y 520.885,Z 860.01,A -85,B 0,C 180,E1 21728.88,E2 21728.88} C_VEL
LIN {X 0,Y 517.058,Z 883.337,A -85,B 0,C 180,E1 21727.908,E2 21727.908} C_VEL
LIN {X 0,Y 512.509,Z 906.563,A -85,B 0,C 180,E1 21726.726,E2 21726.726} C_VEL
LIN {X 0,Y 508.405,Z 925.509,A -85,B 0,C 180,E1 21725.6,E2 21725.6} C_VEL
LIN {X 0,Y 503.92,Z 944.58,A -85,B 0,C 180,E1 21724.298,E2 21724.298} C_VEL
LIN {X 0,Y 498.081,Z 967.406,A -85,B 0,C 180,E1 21722.478,E2 21722.478} C_VEL
LIN {X 0,Y 494.306,Z 981.31,A -85,B 0,C 180,E1 21721.212,E2 21721.212} C_VEL
LIN {X 0,Y 491.871,Z 987.258,A -85,B 0,C 180,E1 21720.703,E2 21720.703} C_VEL
LIN {X 0,Y 482.403,Z 1003.326,A -85,B 0,C 180,E1 21719.511,E2 21719.511} C_VEL
LIN {X 0,Y 480.308,Z 1008.071,A -85,B 0,C 180,E1 21719.015,E2 21719.015} C_VEL
LIN {X 0,Y 475.141,Z 1024.665,A -85,B 0,C 180,E1 21716.9,E2 21716.9} C_VEL
LIN {X 0,Y 470.509,Z 1039.49,A -85,B 0,C 180,E1 21714.748,E2 21714.748} C_VEL
LIN {X 0,Y 465.546,Z 1055.553,A -85,B 0,C 180,E1 21712.077,E2 21712.077} C_VEL
LIN {X 0,Y 461.418,Z 1068.826,A -85,B 0,C 180,E1 21709.494,E2 21709.494} C_VEL
LIN {X 0,Y 458.133,Z 1080.02,A -85,B 0,C 180,E1 21707.005,E2 21707.005} C_VEL
LIN {X 0,Y 454.937,Z 1091.775,A -85,B 0,C 180,E1 21703.99,E2 21703.99} C_VEL
LIN {X 0,Y 452.464,Z 1101.594,A -85,B 0,C 180,E1 21700.955,E2 21700.955} C_VEL
LIN {X 0,Y 450.873,Z 1108.951,A -85,B 0,C 180,E1 21698.288,E2 21698.288} C_VEL
LIN {X 0,Y 449.576,Z 1116.297,A -85,B 0,C 180,E1 21695.104,E2 21695.104} C_VEL
LIN {X 0,Y 448.776,Z 1121.914,A -85,B 0,C 180,E1 21691.915,E2 21691.915} C_VEL
LIN {X 0,Y 448.402,Z 1125.55,A -85,B 0,C 180,E1 21689.233,E2 21689.233} C_VEL
LIN {X 0,Y 448.207,Z 1128.184,A -85,B 0,C 180,E1 21686.547,E2 21686.547} C_VEL
LIN {X 0,Y 448.131,Z 1130.089,A -85,B 0,C 180,E1 21683.337,E2 21683.337} C_VEL
LIN {X 0,Y 448.118,Z 1130.408,A -85,B 0,C 180,E1 21680.237,E2 21680.237} C_VEL
LIN {X 0,Y 448.164,Z 1129.64,A -85,B 0,C 180,E1 21677.502,E2 21677.502} C_VEL
LIN {X 0,Y 448.24,Z 1127.949,A -85,B 0,C 180,E1 21674.871,E2 21674.871} C_VEL
LIN {X 0,Y 448.491,Z 1125.129,A -85,B 0,C 180,E1 21672.082,E2 21672.082} C_VEL
LIN {X 0,Y 449.127,Z 1119.933,A -85,B 0,C 180,E1 21668.528,E2 21668.528} C_VEL
LIN {X 0,Y 450.074,Z 1114.307,A -85,B 0,C 180,E1 21665.625,E2 21665.625} C_VEL
LIN {X 0,Y 451.515,Z 1107.45,A -85,B 0,C 180,E1 21662.717,E2 21662.717} C_VEL
LIN {X 0,Y 454.049,Z 1097.25,A -85,B 0,C 180,E1 21659.188,E2 21659.188} C_VEL
LIN {X 0,Y 456.646,Z 1088.025,A -85,B 0,C 180,E1 21656.511,E2 21656.511} C_VEL
LIN {X 0,Y 460.06,Z 1077.013,A -85,B 0,C 180,E1 21653.739,E2 21653.739} C_VEL
LIN {X 0,Y 464.611,Z 1063.1,A -85,B 0,C 180,E1 21650.751,E2 21650.751} C_VEL
LIN {X 0,Y 469.078,Z 1049.941,A -85,B 0,C 180,E1 21648.315,E2 21648.315} C_VEL
LIN {X 0,Y 474.039,Z 1035.668,A -85,B 0,C 180,E1 21645.995,E2 21645.995} C_VEL
LIN {X 0,Y 480.476,Z 1016.907,A -85,B 0,C 180,E1 21643.373,E2 21643.373} C_VEL
LIN {X 0,Y 485.76,Z 1001.202,A -85,B 0,C 180,E1 21641.476,E2 21641.476} C_VEL
LIN {X 0,Y 491.222,Z 984.504,A -85,B 0,C 180,E1 21639.7,E2 21639.7} C_VEL
LIN {X 0,Y 498.178,Z 961.975,A -85,B 0,C 180,E1 21637.639,E2 21637.639} C_VEL
LIN {X 0,Y 503.565,Z 943.2,A -85,B 0,C 180,E1 21636.174,E2 21636.174} C_VEL
LIN {X 0,Y 508.722,Z 923.933,A -85,B 0,C 180,E1 21634.868,E2 21634.868} C_VEL
LIN {X 0,Y 514.775,Z 898.667,A -85,B 0,C 180,E1 21633.419,E2 21633.419} C_VEL
LIN {X 0,Y 519.158,Z 877.777,A -85,B 0,C 180,E1 21632.426,E2 21632.426} C_VEL
LIN {X 0,Y 522.847,Z 857.768,A -85,B 0,C 180,E1 21631.623,E2 21631.623} C_VEL
LIN {X 0,Y 526.524,Z 834.406,A -85,B 0,C 180,E1 21630.847,E2 21630.847} C_VEL
LIN {X 0,Y 529.544,Z 809.18,A -85,B 0,C 180,E1 21630.204,E2 21630.204} C_VEL
LIN {X 0,Y 531.441,Z 787.553,A -85,B 0,C 180,E1 21629.785,E2 21629.785} C_VEL
LIN {X 0,Y 544.598,Z 553.847,A -85,B 0,C 180,E1 21626.214,E2 21626.214} C_VEL
LIN {X 0,Y 550.459,Z 453.025,A -85,B 0,C 180,E1 21624.666,E2 21624.666} C_VEL
LIN {X 0,Y 540.526,Z 437.665,A -85,B 0,C 180,E1 21622.142,E2 21622.142} C_VEL
LIN {X 0,Y 532.293,Z 425.861,A -85,B 0,C 180,E1 21619.791,E2 21619.791} C_VEL
LIN {X 0,Y 525.545,Z 416.585,A -85,B 0,C 180,E1 21617.609,E2 21617.609} C_VEL
LIN {X 0,Y 521.891,Z 411.746,A -85,B 0,C 180,E1 21616.301,E2 21616.301} C_VEL
LIN {X 0,Y 518.218,Z 406.856,A -85,B 0,C 180,E1 21614.87,E2 21614.87} C_VEL
LIN {X 0,Y 513.977,Z 401.379,A -85,B 0,C 180,E1 21613.042,E2 21613.042} C_VEL
LIN {X 0,Y 510.189,Z 396.666,A -85,B 0,C 180,E1 21611.188,E2 21611.188} C_VEL
LIN {X 0,Y 506.219,Z 391.653,A -85,B 0,C 180,E1 21608.863,E2 21608.863} C_VEL
LIN {X 0,Y 501.913,Z 386.184,A -85,B 0,C 180,E1 21605.487,E2 21605.487} C_VEL
LIN {X 0,Y 498.076,Z 381.927,A -85,B 0,C 180,E1 21599.655,E2 21599.655} C_VEL
LIN {X 0,Y 497.951,Z 381.661,A -85,B 0,C 180,E1 21596.892,E2 21596.892} C_VEL
LIN {X 0,Y 499.154,Z 383.537,A -85,B 0,C 180,E1 21593.559,E2 21593.559} C_VEL
LIN {X 0,Y 502.682,Z 387.079,A -85,B 0,C 180,E1 21589.571,E2 21589.571} C_VEL
LIN {X 0,Y 506.807,Z 392.178,A -85,B 0,C 180,E1 21586.538,E2 21586.538} C_VEL
LIN {X 0,Y 512.13,Z 398.978,A -85,B 0,C 180,E1 21583.613,E2 21583.613} C_VEL
LIN {X 0,Y 516.163,Z 404.027,A -85,B 0,C 180,E1 21581.769,E2 21581.769} C_VEL
LIN {X 0,Y 520.834,Z 410.162,A -85,B 0,C 180,E1 21579.872,E2 21579.872} C_VEL
LIN {X 0,Y 525.533,Z 416.424,A -85,B 0,C 180,E1 21578.163,E2 21578.163} C_VEL
LIN {X 0,Y 532.305,Z 425.786,A -85,B 0,C 180,E1 21575.974,E2 21575.974} C_VEL
LIN {X 0,Y 540.208,Z 437.102,A -85,B 0,C 180,E1 21573.715,E2 21573.715} C_VEL
LIN {X 0,Y 549.156,Z 450.92,A -85,B 0,C 180,E1 21571.418,E2 21571.418} C_VEL
LIN {X 0,Y 552.78,Z 457.107,A -85,B 0,C 180,E1 21570.548,E2 21570.548} C_VEL
LIN {X 0,Y 540.996,Z 664.472,A -85,B 0,C 180,E1 21567.299,E2 21567.299} C_VEL
LIN {X 0,Y 532.578,Z 819.328,A -85,B 0,C 180,E1 21564.875,E2 21564.875} C_VEL
LIN {X 0,Y 529.896,Z 847.065,A -85,B 0,C 180,E1 21564.335,E2 21564.335} C_VEL
LIN {X 0,Y 526.305,Z 872.815,A -85,B 0,C 180,E1 21563.664,E2 21563.664} C_VEL
LIN {X 0,Y 522.848,Z 893.935,A -85,B 0,C 180,E1 21562.977,E2 21562.977} C_VEL
LIN {X 0,Y 518.993,Z 914.571,A -85,B 0,C 180,E1 21562.174,E2 21562.174} C_VEL
LIN {X 0,Y 514.289,Z 937.129,A -85,B 0,C 180,E1 21561.136,E2 21561.136} C_VEL
LIN {X 0,Y 508,Z 964.063,A -85,B 0,C 180,E1 21559.641,E2 21559.641} C_VEL
LIN {X 0,Y 503.004,Z 983.672,A -85,B 0,C 180,E1 21558.366,E2 21558.366} C_VEL
LIN {X 0,Y 497.893,Z 1002.584,A -85,B 0,C 180,E1 21556.968,E2 21556.968} C_VEL
LIN {X 0,Y 492.534,Z 1021.596,A -85,B 0,C 180,E1 21555.379,E2 21555.379} C_VEL
LIN {X 0,Y 485.868,Z 1044.552,A -85,B 0,C 180,E1 21553.176,E2 21553.176} C_VEL
LIN {X 0,Y 479.997,Z 1064.043,A -85,B 0,C 180,E1 21551.008,E2 21551.008} C_VEL
LIN {X 0,Y 475.069,Z 1080.46,A -85,B 0,C 180,E1 21548.952,E2 21548.952} C_VEL
LIN {X 0,Y 470.275,Z 1096.615,A -85,B 0,C 180,E1 21546.687,E2 21546.687} C_VEL
LIN {X 0,Y 464.694,Z 1116.052,A -85,B 0,C 180,E1 21543.571,E2 21543.571} C_VEL
LIN {X 0,Y 460.771,Z 1130.313,A -85,B 0,C 180,E1 21540.95,E2 21540.95} C_VEL
LIN {X 0,Y 457.637,Z 1142.473,A -85,B 0,C 180,E1 21538.444,E2 21538.444} C_VEL
LIN {X 0,Y 454.719,Z 1155.025,A -85,B 0,C 180,E1 21535.529,E2 21535.529} C_VEL
LIN {X 0,Y 452.052,Z 1167.769,A -85,B 0,C 180,E1 21532.061,E2 21532.061} C_VEL
LIN {X 0,Y 450.545,Z 1176.394,A -85,B 0,C 180,E1 21529.309,E2 21529.309} C_VEL
LIN {X 0,Y 449.466,Z 1183.508,A -85,B 0,C 180,E1 21526.677,E2 21526.677} C_VEL
LIN {X 0,Y 448.768,Z 1189.52,A -85,B 0,C 180,E1 21524.055,E2 21524.055} C_VEL
LIN {X 0,Y 448.308,Z 1194.466,A -85,B 0,C 180,E1 21521.449,E2 21521.449} C_VEL
LIN {X 0,Y 448.08,Z 1198.383,A -85,B 0,C 180,E1 21518.857,E2 21518.857} C_VEL
LIN {X 0,Y 447.974,Z 1201.289,A -85,B 0,C 180,E1 21516.279,E2 21516.279} C_VEL
LIN {X 0,Y 447.939,Z 1203.202,A -85,B 0,C 180,E1 21513.712,E2 21513.712} C_VEL
LIN {X 0,Y 447.937,Z 1204.133,A -85,B 0,C 180,E1 21511.151,E2 21511.151} C_VEL
LIN {X 0,Y 447.938,Z 1204.111,A -85,B 0,C 180,E1 21508.721,E2 21508.721} C_VEL
LIN {X 0,Y 447.938,Z 1203.158,A -85,B 0,C 180,E1 21506.201,E2 21506.201} C_VEL
LIN {X 0,Y 447.973,Z 1201.302,A -85,B 0,C 180,E1 21503.721,E2 21503.721} C_VEL
LIN {X 0,Y 448.079,Z 1198.408,A -85,B 0,C 180,E1 21501.143,E2 21501.143} C_VEL
LIN {X 0,Y 448.306,Z 1194.51,A -85,B 0,C 180,E1 21498.551,E2 21498.551} C_VEL
LIN {X 0,Y 448.766,Z 1189.587,A -85,B 0,C 180,E1 21495.945,E2 21495.945} C_VEL
LIN {X 0,Y 449.464,Z 1183.605,A -85,B 0,C 180,E1 21493.324,E2 21493.324} C_VEL
LIN {X 0,Y 450.609,Z 1176.158,A -85,B 0,C 180,E1 21490.559,E2 21490.559} C_VEL
LIN {X 0,Y 452.539,Z 1165.727,A -85,B 0,C 180,E1 21487.254,E2 21487.254} C_VEL
LIN {X 0,Y 455.103,Z 1153.695,A -85,B 0,C 180,E1 21484.075,E2 21484.075} C_VEL
LIN {X 0,Y 457.668,Z 1142.87,A -85,B 0,C 180,E1 21481.559,E2 21481.559} C_VEL
LIN {X 0,Y 460.627,Z 1131.402,A -85,B 0,C 180,E1 21479.185,E2 21479.185} C_VEL
LIN {X 0,Y 464.107,Z 1118.628,A -85,B 0,C 180,E1 21476.824,E2 21476.824} C_VEL
LIN {X 0,Y 468.566,Z 1102.781,A -85,B 0,C 180,E1 21474.22,E2 21474.22} C_VEL
LIN {X 0,Y 474.027,Z 1083.657,A -85,B 0,C 180,E1 21471.497,E2 21471.497} C_VEL
LIN {X 0,Y 478.799,Z 1067.05,A -85,B 0,C 180,E1 21469.421,E2 21469.421} C_VEL
LIN {X 0,Y 483.483,Z 1050.616,A -85,B 0,C 180,E1 21467.588,E2 21467.588} C_VEL
LIN {X 0,Y 488.696,Z 1031.951,A -85,B 0,C 180,E1 21465.735,E2 21465.735} C_VEL
LIN {X 0,Y 495.262,Z 1007.475,A -85,B 0,C 180,E1 21463.635,E2 21463.635} C_VEL
LIN {X 0,Y 500.105,Z 988.24,A -85,B 0,C 180,E1 21462.205,E2 21462.205} C_VEL
LIN {X 0,Y 504.754,Z 968.592,A -85,B 0,C 180,E1 21460.919,E2 21460.919} C_VEL
LIN {X 0,Y 509.271,Z 948.161,A -85,B 0,C 180,E1 21459.751,E2 21459.751} C_VEL
LIN {X 0,Y 514.48,Z 922.314,A -85,B 0,C 180,E1 21458.49,E2 21458.49} C_VEL
LIN {X 0,Y 518.713,Z 897.804,A -85,B 0,C 180,E1 21457.515,E2 21457.515} C_VEL
LIN {X 0,Y 522.002,Z 876.158,A -85,B 0,C 180,E1 21456.802,E2 21456.802} C_VEL
LIN {X 0,Y 524.79,Z 854.451,A -85,B 0,C 180,E1 21456.216,E2 21456.216} C_VEL
LIN {X 0,Y 527.595,Z 827.02,A -85,B 0,C 180,E1 21455.641,E2 21455.641} C_VEL
LIN {X 0,Y 529.962,Z 780.365,A -85,B 0,C 180,E1 21454.908,E2 21454.908} C_VEL
LIN {X 0,Y 540.137,Z 556.59,A -85,B 0,C 180,E1 21451.512,E2 21451.512} C_VEL
LIN {X 0,Y 544.926,Z 454.736,A -85,B 0,C 180,E1 21449.94,E2 21449.94} C_VEL
LIN {X 0,Y 530.155,Z 432.124,A -85,B 0,C 180,E1 21447.096,E2 21447.096} C_VEL
LIN {X 0,Y 518.444,Z 414.985,A -85,B 0,C 180,E1 21444.589,E2 21444.589} C_VEL
LIN {X 0,Y 507.865,Z 400.336,A -85,B 0,C 180,E1 21442.089,E2 21442.089} C_VEL
LIN {X 0,Y 499.407,Z 389.182,A -85,B 0,C 180,E1 21439.869,E2 21439.869} C_VEL
LIN {X 0,Y 495.246,Z 383.809,A -85,B 0,C 180,E1 21438.694,E2 21438.694} C_VEL
LIN {X 0,Y 487.848,Z 374.503,A -85,B 0,C 180,E1 21436.43,E2 21436.43} C_VEL
LIN {X 0,Y 483.224,Z 368.839,A -85,B 0,C 180,E1 21434.867,E2 21434.867} C_VEL
LIN {X 0,Y 478.768,Z 363.359,A -85,B 0,C 180,E1 21433.22,E2 21433.22} C_VEL
LIN {X 0,Y 474.921,Z 358.97,A -85,B 0,C 180,E1 21431.692,E2 21431.692} C_VEL
LIN {X 0,Y 472.67,Z 356.458,A -85,B 0,C 180,E1 21430.729,E2 21430.729} C_VEL
LIN {X 0,Y 468.433,Z 351.487,A -85,B 0,C 180,E1 21428.717,E2 21428.717} C_VEL
LIN {X 0,Y 465.412,Z 347.963,A -85,B 0,C 180,E1 21426.91,E2 21426.91} C_VEL
LIN {X 0,Y 464.532,Z 345.941,A -85,B 0,C 180,E1 21425.806,E2 21425.806} C_VEL
LIN {X 0,Y 461.691,Z 341.575,A -85,B 0,C 180,E1 21422.358,E2 21422.358} C_VEL
LIN {X 0,Y 460.95,Z 340.235,A -85,B 0,C 180,E1 21421.119,E2 21421.119} C_VEL
LIN {X 0,Y 458.53,Z 337.135,A -85,B 0,C 180,E1 21415.497,E2 21415.497} C_VEL
LIN {X 0,Y 458.352,Z 336.698,A -85,B 0,C 180,E1 21412.101,E2 21412.101} C_VEL
LIN {X 0,Y 458.883,Z 337.873,A -85,B 0,C 180,E1 21408.436,E2 21408.436} C_VEL
LIN {X 0,Y 461.253,Z 340.777,A -85,B 0,C 180,E1 21403.799,E2 21403.799} C_VEL
LIN {X 0,Y 463.636,Z 345.176,A -85,B 0,C 180,E1 21400.34,E2 21400.34} C_VEL
LIN {X 0,Y 464.593,Z 346.569,A -85,B 0,C 180,E1 21399.331,E2 21399.331} C_VEL
LIN {X 0,Y 466.264,Z 349.509,A -85,B 0,C 180,E1 21397.958,E2 21397.958} C_VEL
LIN {X 0,Y 469.336,Z 352.61,A -85,B 0,C 180,E1 21396.389,E2 21396.389} C_VEL
LIN {X 0,Y 474.543,Z 358.665,A -85,B 0,C 180,E1 21394.006,E2 21394.006} C_VEL
LIN {X 0,Y 479.598,Z 364.645,A -85,B 0,C 180,E1 21391.991,E2 21391.991} C_VEL
LIN {X 0,Y 484.652,Z 370.754,A -85,B 0,C 180,E1 21390.184,E2 21390.184} C_VEL
LIN {X 0,Y 490.826,Z 378.461,A -85,B 0,C 180,E1 21388.189,E2 21388.189} C_VEL
LIN {X 0,Y 497.399,Z 386.894,A -85,B 0,C 180,E1 21386.266,E2 21386.266} C_VEL
LIN {X 0,Y 504.319,Z 395.83,A -85,B 0,C 180,E1 21384.415,E2 21384.415} C_VEL
LIN {X 0,Y 514.636,Z 410.203,A -85,B 0,C 180,E1 21381.881,E2 21381.881} C_VEL
LIN {X 0,Y 525.891,Z 426.467,A -85,B 0,C 180,E1 21379.403,E2 21379.403} C_VEL
LIN {X 0,Y 537.312,Z 444.154,A -85,B 0,C 180,E1 21377.107,E2 21377.107} C_VEL
LIN {X 0,Y 539.988,Z 448.704,A -85,B 0,C 180,E1 21376.591,E2 21376.591} C_VEL
LIN {X 0,Y 529.063,Z 675.429,A -85,B 0,C 180,E1 21373.188,E2 21373.188} C_VEL
LIN {X 0,Y 523.62,Z 789.217,A -85,B 0,C 180,E1 21371.464,E2 21371.464} C_VEL
LIN {X 0,Y 521.324,Z 815.989,A -85,B 0,C 180,E1 21370.917,E2 21370.917} C_VEL
LIN {X 0,Y 518.445,Z 839.95,A -85,B 0,C 180,E1 21370.246,E2 21370.246} C_VEL
LIN {X 0,Y 515.515,Z 860.226,A -85,B 0,C 180,E1 21369.542,E2 21369.542} C_VEL
LIN {X 0,Y 511.79,Z 882.352,A -85,B 0,C 180,E1 21368.623,E2 21368.623} C_VEL
LIN {X 0,Y 506.986,Z 906.47,A -85,B 0,C 180,E1 21367.403,E2 21367.403} C_VEL
LIN {X 0,Y 502.753,Z 925.448,A -85,B 0,C 180,E1 21366.275,E2 21366.275} C_VEL
LIN {X 0,Y 498.3,Z 943.83,A -85,B 0,C 180,E1 21365.02,E2 21365.02} C_VEL
LIN {X 0,Y 492.689,Z 965.461,A -85,B 0,C 180,E1 21363.316,E2 21363.316} C_VEL
LIN {X 0,Y 487.104,Z 985.124,A -85,B 0,C 180,E1 21361.493,E2 21361.493} C_VEL
LIN {X 0,Y 482.333,Z 1001.281,A -85,B 0,C 180,E1 21359.788,E2 21359.788} C_VEL
LIN {X 0,Y 480.308,Z 1008.071,A -85,B 0,C 180,E1 21359.015,E2 21359.015} C_VEL
LIN {X 0,Y 477.771,Z 1013.562,A -85,B 0,C 180,E1 21358.426,E2 21358.426} C_VEL
LIN {X 0,Y 468.605,Z 1027.611,A -85,B 0,C 180,E1 21357.081,E2 21357.081} C_VEL
LIN {X 0,Y 466.152,Z 1032.679,A -85,B 0,C 180,E1 21356.432,E2 21356.432} C_VEL
LIN {X 0,Y 460.942,Z 1048.476,A -85,B 0,C 180,E1 21353.931,E2 21353.931} C_VEL
LIN {X 0,Y 456.721,Z 1061.484,A -85,B 0,C 180,E1 21351.579,E2 21351.579} C_VEL
LIN {X 0,Y 452.398,Z 1075.415,A -85,B 0,C 180,E1 21348.691,E2 21348.691} C_VEL
LIN {X 0,Y 448.742,Z 1087.461,A -85,B 0,C 180,E1 21345.721,E2 21345.721} C_VEL
LIN {X 0,Y 446.194,Z 1096.726,A -85,B 0,C 180,E1 21343.081,E2 21343.081} C_VEL
LIN {X 0,Y 443.831,Z 1106.382,A -85,B 0,C 180,E1 21339.858,E2 21339.858} C_VEL
LIN {X 0,Y 442.235,Z 1113.899,A -85,B 0,C 180,E1 21336.752,E2 21336.752} C_VEL
LIN {X 0,Y 441.299,Z 1119.35,A -85,B 0,C 180,E1 21334.028,E2 21334.028} C_VEL
LIN {X 0,Y 440.67,Z 1123.94,A -85,B 0,C 180,E1 21331.17,E2 21331.17} C_VEL
LIN {X 0,Y 440.312,Z 1128.001,A -85,B 0,C 180,E1 21327.657,E2 21327.657} C_VEL
LIN {X 0,Y 440.181,Z 1130.036,A -85,B 0,C 180,E1 21324.787,E2 21324.787} C_VEL
LIN {X 0,Y 440.165,Z 1130.978,A -85,B 0,C 180,E1 21322.035,E2 21322.035} C_VEL
LIN {X 0,Y 440.149,Z 1130.928,A -85,B 0,C 180,E1 21319.265,E2 21319.265} C_VEL
LIN {X 0,Y 440.241,Z 1129.568,A -85,B 0,C 180,E1 21315.935,E2 21315.935} C_VEL
LIN {X 0,Y 440.457,Z 1126.849,A -85,B 0,C 180,E1 21312.836,E2 21312.836} C_VEL
LIN {X 0,Y 440.842,Z 1123.449,A -85,B 0,C 180,E1 21310.11,E2 21310.11} C_VEL
LIN {X 0,Y 441.565,Z 1118.76,A -85,B 0,C 180,E1 21307.219,E2 21307.219} C_VEL
LIN {X 0,Y 443.026,Z 1111.585,A -85,B 0,C 180,E1 21303.746,E2 21303.746} C_VEL
LIN {X 0,Y 444.958,Z 1103.625,A -85,B 0,C 180,E1 21300.668,E2 21300.668} C_VEL
LIN {X 0,Y 447.359,Z 1095.085,A -85,B 0,C 180,E1 21297.864,E2 21297.864} C_VEL
LIN {X 0,Y 451.287,Z 1082.572,A -85,B 0,C 180,E1 21294.404,E2 21294.404} C_VEL
LIN {X 0,Y 455.152,Z 1071.101,A -85,B 0,C 180,E1 21291.721,E2 21291.721} C_VEL
LIN {X 0,Y 459.694,Z 1058.285,A -85,B 0,C 180,E1 21289.104,E2 21289.104} C_VEL
LIN {X 0,Y 465.558,Z 1041.938,A -85,B 0,C 180,E1 21286.247,E2 21286.247} C_VEL
LIN {X 0,Y 470.827,Z 1027.315,A -85,B 0,C 180,E1 21284.041,E2 21284.041} C_VEL
LIN {X 0,Y 476.694,Z 1010.94,A -85,B 0,C 180,E1 21281.875,E2 21281.875} C_VEL
LIN {X 0,Y 483.528,Z 991.073,A -85,B 0,C 180,E1 21279.622,E2 21279.622} C_VEL
LIN {X 0,Y 488.994,Z 974.422,A -85,B 0,C 180,E1 21277.987,E2 21277.987} C_VEL
LIN {X 0,Y 494.441,Z 956.964,A -85,B 0,C 180,E1 21276.481,E2 21276.481} C_VEL
LIN {X 0,Y 500.8,Z 935.262,A -85,B 0,C 180,E1 21274.858,E2 21274.858} C_VEL
LIN {X 0,Y 506.493,Z 913.337,A -85,B 0,C 180,E1 21273.483,E2 21273.483} C_VEL
LIN {X 0,Y 511.027,Z 894.081,A -85,B 0,C 180,E1 21272.445,E2 21272.445} C_VEL
LIN {X 0,Y 515.922,Z 870.849,A -85,B 0,C 180,E1 21271.385,E2 21271.385} C_VEL
LIN {X 0,Y 520.328,Z 845.369,A -85,B 0,C 180,E1 21270.45,E2 21270.45} C_VEL
LIN {X 0,Y 523.403,Z 823.685,A -85,B 0,C 180,E1 21269.815,E2 21269.815} C_VEL
LIN {X 0,Y 526.133,Z 799.577,A -85,B 0,C 180,E1 21269.268,E2 21269.268} C_VEL
LIN {X 0,Y 528.541,Z 763.997,A -85,B 0,C 180,E1 21268.682,E2 21268.682} C_VEL
LIN {X 0,Y 542.274,Z 527.144,A -85,B 0,C 180,E1 21265.065,E2 21265.065} C_VEL
LIN {X 0,Y 546.428,Z 457.692,A -85,B 0,C 180,E1 21263.987,E2 21263.987} C_VEL
LIN {X 0,Y 537.518,Z 443.688,A -85,B 0,C 180,E1 21261.641,E2 21261.641} C_VEL
LIN {X 0,Y 528.67,Z 430.905,A -85,B 0,C 180,E1 21259.013,E2 21259.013} C_VEL
LIN {X 0,Y 522.906,Z 422.923,A -85,B 0,C 180,E1 21257.069,E2 21257.069} C_VEL
LIN {X 0,Y 517.099,Z 414.975,A -85,B 0,C 180,E1 21254.845,E2 21254.845} C_VEL
LIN {X 0,Y 512.277,Z 408.803,A -85,B 0,C 180,E1 21252.742,E2 21252.742} C_VEL
LIN {X 0,Y 508.792,Z 404.35,A -85,B 0,C 180,E1 21250.989,E2 21250.989} C_VEL
LIN {X 0,Y 505.068,Z 399.527,A -85,B 0,C 180,E1 21248.768,E2 21248.768} C_VEL
LIN {X 0,Y 500.807,Z 394.06,A -85,B 0,C 180,E1 21245.384,E2 21245.384} C_VEL
LIN {X 0,Y 497.096,Z 389.875,A -85,B 0,C 180,E1 21239.654,E2 21239.654} C_VEL
LIN {X 0,Y 496.965,Z 389.604,A -85,B 0,C 180,E1 21236.886,E2 21236.886} C_VEL
LIN {X 0,Y 498.237,Z 391.603,A -85,B 0,C 180,E1 21233.431,E2 21233.431} C_VEL
LIN {X 0,Y 501.508,Z 394.884,A -85,B 0,C 180,E1 21229.721,E2 21229.721} C_VEL
LIN {X 0,Y 506.17,Z 400.883,A -85,B 0,C 180,E1 21226.288,E2 21226.288} C_VEL
LIN {X 0,Y 510.693,Z 406.686,A -85,B 0,C 180,E1 21223.799,E2 21223.799} C_VEL
LIN {X 0,Y 514.669,Z 411.773,A -85,B 0,C 180,E1 21221.948,E2 21221.948} C_VEL
LIN {X 0,Y 519.148,Z 417.731,A -85,B 0,C 180,E1 21220.097,E2 21220.097} C_VEL
LIN {X 0,Y 524.002,Z 424.296,A -85,B 0,C 180,E1 21218.305,E2 21218.305} C_VEL
LIN {X 0,Y 531.738,Z 435.066,A -85,B 0,C 180,E1 21215.799,E2 21215.799} C_VEL
LIN {X 0,Y 540.657,Z 448.469,A -85,B 0,C 180,E1 21213.265,E2 21213.265} C_VEL
LIN {X 0,Y 548.702,Z 461.423,A -85,B 0,C 180,E1 21211.216,E2 21211.216} C_VEL
LIN {X 0,Y 536.534,Z 668.644,A -85,B 0,C 180,E1 21207.96,E2 21207.96} C_VEL
LIN {X 0,Y 528.06,Z 819.007,A -85,B 0,C 180,E1 21205.596,E2 21205.596} C_VEL
LIN {X 0,Y 525.298,Z 846.755,A -85,B 0,C 180,E1 21205.056,E2 21205.056} C_VEL
LIN {X 0,Y 521.616,Z 872.415,A -85,B 0,C 180,E1 21204.388,E2 21204.388} C_VEL
LIN {X 0,Y 518.148,Z 893.02,A -85,B 0,C 180,E1 21203.719,E2 21203.719} C_VEL
LIN {X 0,Y 514.209,Z 913.439,A -85,B 0,C 180,E1 21202.929,E2 21202.929} C_VEL
LIN {X 0,Y 509.605,Z 934.942,A -85,B 0,C 180,E1 21201.946,E2 21201.946} C_VEL
LIN {X 0,Y 503.367,Z 961.148,A -85,B 0,C 180,E1 21200.515,E2 21200.515} C_VEL
LIN {X 0,Y 497.741,Z 982.424,A -85,B 0,C 180,E1 21199.14,E2 21199.14} C_VEL
LIN {X 0,Y 492.432,Z 1001.387,A -85,B 0,C 180,E1 21197.74,E2 21197.74} C_VEL
LIN {X 0,Y 487.026,Z 1019.818,A -85,B 0,C 180,E1 21196.197,E2 21196.197} C_VEL
LIN {X 0,Y 480.458,Z 1041.703,A -85,B 0,C 180,E1 21194.111,E2 21194.111} C_VEL
LIN {X 0,Y 473.789,Z 1062.933,A -85,B 0,C 180,E1 21191.744,E2 21191.744} C_VEL
LIN {X 0,Y 468.721,Z 1079.065,A -85,B 0,C 180,E1 21189.709,E2 21189.709} C_VEL
LIN {X 0,Y 463.746,Z 1095.078,A -85,B 0,C 180,E1 21187.445,E2 21187.445} C_VEL
LIN {X 0,Y 458.268,Z 1113.131,A -85,B 0,C 180,E1 21184.56,E2 21184.56} C_VEL
LIN {X 0,Y 453.686,Z 1128.897,A -85,B 0,C 180,E1 21181.636,E2 21181.636} C_VEL
LIN {X 0,Y 450.349,Z 1141.09,A -85,B 0,C 180,E1 21179.093,E2 21179.093} C_VEL
LIN {X 0,Y 447.428,Z 1152.803,A -85,B 0,C 180,E1 21176.345,E2 21176.345} C_VEL
LIN {X 0,Y 444.607,Z 1165.604,A -85,B 0,C 180,E1 21172.896,E2 21172.896} C_VEL
LIN {X 0,Y 442.765,Z 1175.26,A -85,B 0,C 180,E1 21169.8,E2 21169.8} C_VEL
LIN {X 0,Y 441.572,Z 1182.777,A -85,B 0,C 180,E1 21166.984,E2 21166.984} C_VEL
LIN {X 0,Y 440.826,Z 1188.808,A -85,B 0,C 180,E1 21164.314,E2 21164.314} C_VEL
LIN {X 0,Y 440.345,Z 1193.772,A -85,B 0,C 180,E1 21161.659,E2 21161.659} C_VEL
LIN {X 0,Y 440.104,Z 1197.7,A -85,B 0,C 180,E1 21159.019,E2 21159.019} C_VEL
LIN {X 0,Y 439.998,Z 1200.616,A -85,B 0,C 180,E1 21156.393,E2 21156.393} C_VEL
LIN {X 0,Y 439.963,Z 1202.48,A -85,B 0,C 180,E1 21153.88,E2 21153.88} C_VEL
LIN {X 0,Y 439.964,Z 1203.424,A -85,B 0,C 180,E1 21151.433,E2 21151.433} C_VEL
LIN {X 0,Y 439.961,Z 1203.502,A -85,B 0,C 180,E1 21148.958,E2 21148.958} C_VEL
LIN {X 0,Y 439.962,Z 1202.625,A -85,B 0,C 180,E1 21146.352,E2 21146.352} C_VEL
LIN {X 0,Y 439.991,Z 1200.765,A -85,B 0,C 180,E1 21143.738,E2 21143.738} C_VEL
LIN {X 0,Y 440.093,Z 1197.915,A -85,B 0,C 180,E1 21141.113,E2 21141.113} C_VEL
LIN {X 0,Y 440.323,Z 1194.059,A -85,B 0,C 180,E1 21138.473,E2 21138.473} C_VEL
LIN {X 0,Y 440.793,Z 1189.177,A -85,B 0,C 180,E1 21135.82,E2 21135.82} C_VEL
LIN {X 0,Y 441.519,Z 1183.236,A -85,B 0,C 180,E1 21133.15,E2 21133.15} C_VEL
LIN {X 0,Y 442.685,Z 1175.925,A -85,B 0,C 180,E1 21130.37,E2 21130.37} C_VEL
LIN {X 0,Y 444.422,Z 1166.734,A -85,B 0,C 180,E1 21127.374,E2 21127.374} C_VEL
LIN {X 0,Y 447.259,Z 1154.029,A -85,B 0,C 180,E1 21123.871,E2 21123.871} C_VEL
LIN {X 0,Y 450.208,Z 1142.107,A -85,B 0,C 180,E1 21121.052,E2 21121.052} C_VEL
LIN {X 0,Y 453.528,Z 1129.879,A -85,B 0,C 180,E1 21118.5,E2 21118.5} C_VEL
LIN {X 0,Y 457.612,Z 1115.485,A -85,B 0,C 180,E1 21115.838,E2 21115.838} C_VEL
LIN {X 0,Y 463.199,Z 1096.499,A -85,B 0,C 180,E1 21112.802,E2 21112.802} C_VEL
LIN {X 0,Y 467.888,Z 1080.766,A -85,B 0,C 180,E1 21110.604,E2 21110.604} C_VEL
LIN {X 0,Y 472.645,Z 1064.84,A -85,B 0,C 180,E1 21108.618,E2 21108.618} C_VEL
LIN {X 0,Y 477.851,Z 1047.212,A -85,B 0,C 180,E1 21106.662,E2 21106.662} C_VEL
LIN {X 0,Y 484.589,Z 1023.614,A -85,B 0,C 180,E1 21104.386,E2 21104.386} C_VEL
LIN {X 0,Y 489.806,Z 1004.449,A -85,B 0,C 180,E1 21102.789,E2 21102.789} C_VEL
LIN {X 0,Y 494.637,Z 985.801,A -85,B 0,C 180,E1 21101.415,E2 21101.415} C_VEL
LIN {X 0,Y 499.389,Z 966.265,A -85,B 0,C 180,E1 21100.145,E2 21100.145} C_VEL
LIN {X 0,Y 505.045,Z 941.189,A -85,B 0,C 180,E1 21098.738,E2 21098.738} C_VEL
LIN {X 0,Y 509.873,Z 916.663,A -85,B 0,C 180,E1 21097.605,E2 21097.605} C_VEL
LIN {X 0,Y 513.632,Z 895.262,A -85,B 0,C 180,E1 21096.77,E2 21096.77} C_VEL
LIN {X 0,Y 516.94,Z 873.834,A -85,B 0,C 180,E1 21096.075,E2 21096.075} C_VEL
LIN {X 0,Y 520.207,Z 848.702,A -85,B 0,C 180,E1 21095.418,E2 21095.418} C_VEL
LIN {X 0,Y 522.772,Z 820.532,A -85,B 0,C 180,E1 21094.87,E2 21094.87} C_VEL
LIN {X 0,Y 528.153,Z 707.956,A -85,B 0,C 180,E1 21093.139,E2 21093.139} C_VEL
LIN {X 0,Y 538.632,Z 489.54,A -85,B 0,C 180,E1 21089.794,E2 21089.794} C_VEL
LIN {X 0,Y 540.034,Z 458.848,A -85,B 0,C 180,E1 21089.303,E2 21089.303} C_VEL
LIN {X 0,Y 526.751,Z 438.281,A -85,B 0,C 180,E1 21086.675,E2 21086.675} C_VEL
LIN {X 0,Y 515.516,Z 421.651,A -85,B 0,C 180,E1 21084.219,E2 21084.219} C_VEL
LIN {X 0,Y 505.084,Z 407.024,A -85,B 0,C 180,E1 21081.697,E2 21081.697} C_VEL
LIN {X 0,Y 496.744,Z 395.895,A -85,B 0,C 180,E1 21079.459,E2 21079.459} C_VEL
LIN {X 0,Y 492.83,Z 390.787,A -85,B 0,C 180,E1 21078.329,E2 21078.329} C_VEL
LIN {X 0,Y 485.637,Z 381.634,A -85,B 0,C 180,E1 21076.077,E2 21076.077} C_VEL
LIN {X 0,Y 481.412,Z 376.342,A -85,B 0,C 180,E1 21074.617,E2 21074.617} C_VEL
LIN {X 0,Y 476.852,Z 370.747,A -85,B 0,C 180,E1 21072.904,E2 21072.904} C_VEL
LIN {X 0,Y 473.019,Z 366.174,A -85,B 0,C 180,E1 21071.338,E2 21071.338} C_VEL
LIN {X 0,Y 466.958,Z 359.156,A -85,B 0,C 180,E1 21068.497,E2 21068.497} C_VEL
LIN {X 0,Y 461.882,Z 353.368,A -85,B 0,C 180,E1 21065.59,E2 21065.59} C_VEL
LIN {X 0,Y 457.788,Z 348.869,A -85,B 0,C 180,E1 21062.566,E2 21062.566} C_VEL
LIN {X 0,Y 456.896,Z 347.161,A -85,B 0,C 180,E1 21061.254,E2 21061.254} C_VEL
LIN {X 0,Y 454.389,Z 343.958,A -85,B 0,C 180,E1 21055.414,E2 21055.414} C_VEL
LIN {X 0,Y 454.227,Z 343.55,A -85,B 0,C 180,E1 21052.118,E2 21052.118} C_VEL
LIN {X 0,Y 454.697,Z 344.69,A -85,B 0,C 180,E1 21048.456,E2 21048.456} C_VEL
LIN {X 0,Y 457.027,Z 347.56,A -85,B 0,C 180,E1 21043.868,E2 21043.868} C_VEL
LIN {X 0,Y 460.516,Z 352.244,A -85,B 0,C 180,E1 21040.814,E2 21040.814} C_VEL
LIN {X 0,Y 462.593,Z 354.199,A -85,B 0,C 180,E1 21039.503,E2 21039.503} C_VEL
LIN {X 0,Y 466.739,Z 358.99,A -85,B 0,C 180,E1 21037.185,E2 21037.185} C_VEL
LIN {X 0,Y 472.872,Z 366.183,A -85,B 0,C 180,E1 21034.272,E2 21034.272} C_VEL
LIN {X 0,Y 477.749,Z 372.035,A -85,B 0,C 180,E1 21032.285,E2 21032.285} C_VEL
LIN {X 0,Y 482.739,Z 378.168,A -85,B 0,C 180,E1 21030.464,E2 21030.464} C_VEL
LIN {X 0,Y 490.094,Z 387.405,A -85,B 0,C 180,E1 21028.07,E2 21028.07} C_VEL
LIN {X 0,Y 498.85,Z 398.918,A -85,B 0,C 180,E1 21025.546,E2 21025.546} C_VEL
LIN {X 0,Y 508.526,Z 412.203,A -85,B 0,C 180,E1 21023.045,E2 21023.045} C_VEL
LIN {X 0,Y 519.374,Z 427.903,A -85,B 0,C 180,E1 21020.521,E2 21020.521} C_VEL
LIN {X 0,Y 531.28,Z 446.218,A -85,B 0,C 180,E1 21018.02,E2 21018.02} C_VEL
LIN {X 0,Y 535.225,Z 452.792,A -85,B 0,C 180,E1 21017.234,E2 21017.234} C_VEL
LIN {X 0,Y 523.887,Z 680.728,A -85,B 0,C 180,E1 21013.797,E2 21013.797} C_VEL
LIN {X 0,Y 518.498,Z 789.67,A -85,B 0,C 180,E1 21012.138,E2 21012.138} C_VEL
LIN {X 0,Y 516.116,Z 816.638,A -85,B 0,C 180,E1 21011.584,E2 21011.584} C_VEL
LIN {X 0,Y 513.184,Z 840.405,A -85,B 0,C 180,E1 21010.915,E2 21010.915} C_VEL
LIN {X 0,Y 510.213,Z 860.42,A -85,B 0,C 180,E1 21010.219,E2 21010.219} C_VEL
LIN {X 0,Y 506.248,Z 883.326,A -85,B 0,C 180,E1 21009.263,E2 21009.263} C_VEL
LIN {X 0,Y 501.328,Z 907.248,A -85,B 0,C 180,E1 21008.045,E2 21008.045} C_VEL
LIN {X 0,Y 496.971,Z 926.224,A -85,B 0,C 180,E1 21006.909,E2 21006.909} C_VEL
LIN {X 0,Y 492.193,Z 945.355,A -85,B 0,C 180,E1 21005.592,E2 21005.592} C_VEL
LIN {X 0,Y 485.978,Z 968.263,A -85,B 0,C 180,E1 21003.745,E2 21003.745} C_VEL
LIN {X 0,Y 480.828,Z 985.855,A -85,B 0,C 180,E1 21002.093,E2 21002.093} C_VEL
LIN {X 0,Y 475.861,Z 1002.119,A -85,B 0,C 180,E1 21000.36,E2 21000.36} C_VEL
LIN {X 0,Y 470.209,Z 1020.166,A -85,B 0,C 180,E1 20998.168,E2 20998.168} C_VEL
LIN {X 0,Y 466.152,Z 1032.679,A -85,B 0,C 180,E1 20996.432,E2 20996.432} C_VEL
LIN {X 0,Y 463.677,Z 1037.704,A -85,B 0,C 180,E1 20995.761,E2 20995.761} C_VEL
LIN {X 0,Y 454.433,Z 1050.353,A -85,B 0,C 180,E1 20994.182,E2 20994.182} C_VEL
LIN {X 0,Y 452.093,Z 1054.945,A -85,B 0,C 180,E1 20993.456,E2 20993.456} C_VEL
LIN {X 0,Y 447.14,Z 1069.653,A -85,B 0,C 180,E1 20990.553,E2 20990.553} C_VEL
LIN {X 0,Y 443.493,Z 1080.906,A -85,B 0,C 180,E1 20987.991,E2 20987.991} C_VEL
LIN {X 0,Y 439.961,Z 1092.744,A -85,B 0,C 180,E1 20984.88,E2 20984.88} C_VEL
LIN {X 0,Y 437.182,Z 1102.615,A -85,B 0,C 180,E1 20981.744,E2 20981.744} C_VEL
LIN {X 0,Y 435.382,Z 1110.01,A -85,B 0,C 180,E1 20978.984,E2 20978.984} C_VEL
LIN {X 0,Y 433.94,Z 1117.114,A -85,B 0,C 180,E1 20975.819,E2 20975.819} C_VEL
LIN {X 0,Y 432.96,Z 1123.075,A -85,B 0,C 180,E1 20972.382,E2 20972.382} C_VEL
LIN {X 0,Y 432.498,Z 1126.892,A -85,B 0,C 180,E1 20969.47,E2 20969.47} C_VEL
LIN {X 0,Y 432.276,Z 1129.516,A -85,B 0,C 180,E1 20966.685,E2 20966.685} C_VEL
LIN {X 0,Y 432.187,Z 1131.411,A -85,B 0,C 180,E1 20963.357,E2 20963.357} C_VEL
LIN {X 0,Y 432.173,Z 1131.723,A -85,B 0,C 180,E1 20960.142,E2 20960.142} C_VEL
LIN {X 0,Y 432.229,Z 1130.958,A -85,B 0,C 180,E1 20957.305,E2 20957.305} C_VEL
LIN {X 0,Y 432.336,Z 1129.273,A -85,B 0,C 180,E1 20954.576,E2 20954.576} C_VEL
LIN {X 0,Y 432.641,Z 1126.466,A -85,B 0,C 180,E1 20951.681,E2 20951.681} C_VEL
LIN {X 0,Y 433.389,Z 1121.379,A -85,B 0,C 180,E1 20948.045,E2 20948.045} C_VEL
LIN {X 0,Y 434.474,Z 1115.846,A -85,B 0,C 180,E1 20945.06,E2 20945.06} C_VEL
LIN {X 0,Y 436.064,Z 1109.198,A -85,B 0,C 180,E1 20942.111,E2 20942.111} C_VEL
LIN {X 0,Y 438.837,Z 1099.426,A -85,B 0,C 180,E1 20938.55,E2 20938.55} C_VEL
LIN {X 0,Y 441.802,Z 1090.007,A -85,B 0,C 180,E1 20935.698,E2 20935.698} C_VEL
LIN {X 0,Y 445.326,Z 1079.756,A -85,B 0,C 180,E1 20933.007,E2 20933.007} C_VEL
LIN {X 0,Y 450.307,Z 1066.094,A -85,B 0,C 180,E1 20929.916,E2 20929.916} C_VEL
LIN {X 0,Y 455.41,Z 1052.359,A -85,B 0,C 180,E1 20927.28,E2 20927.28} C_VEL
LIN {X 0,Y 460.35,Z 1039.293,A -85,B 0,C 180,E1 20925.079,E2 20925.079} C_VEL
LIN {X 0,Y 466.873,Z 1022.114,A -85,B 0,C 180,E1 20922.548,E2 20922.548} C_VEL
LIN {X 0,Y 473.531,Z 1003.716,A -85,B 0,C 180,E1 20920.251,E2 20920.251} C_VEL
LIN {X 0,Y 479.169,Z 987.739,A -85,B 0,C 180,E1 20918.511,E2 20918.511} C_VEL
LIN {X 0,Y 485.874,Z 967.93,A -85,B 0,C 180,E1 20916.624,E2 20916.624} C_VEL
LIN {X 0,Y 492.503,Z 946.465,A -85,B 0,C 180,E1 20914.897,E2 20914.897} C_VEL
LIN {X 0,Y 497.752,Z 928.203,A -85,B 0,C 180,E1 20913.631,E2 20913.631} C_VEL
LIN {X 0,Y 502.924,Z 908.61,A -85,B 0,C 180,E1 20912.452,E2 20912.452} C_VEL
LIN {X 0,Y 508.734,Z 883.735,A -85,B 0,C 180,E1 20911.192,E2 20911.192} C_VEL
LIN {X 0,Y 513.01,Z 862.237,A -85,B 0,C 180,E1 20910.299,E2 20910.299} C_VEL
LIN {X 0,Y 516.379,Z 842.489,A -85,B 0,C 180,E1 20909.612,E2 20909.612} C_VEL
LIN {X 0,Y 519.648,Z 819.359,A -85,B 0,C 180,E1 20908.957,E2 20908.957} C_VEL
LIN {X 0,Y 522.479,Z 792.003,A -85,B 0,C 180,E1 20908.387,E2 20908.387} C_VEL
LIN {X 0,Y 527.727,Z 705.198,A -85,B 0,C 180,E1 20907.038,E2 20907.038} C_VEL
LIN {X 0,Y 542.046,Z 470.95,A -85,B 0,C 180,E1 20903.454,E2 20903.454} C_VEL
LIN {X 0,Y 542.55,Z 462.394,A -85,B 0,C 180,E1 20903.314,E2 20903.314} C_VEL
LIN {X 0,Y 534.015,Z 449.042,A -85,B 0,C 180,E1 20900.983,E2 20900.983} C_VEL
LIN {X 0,Y 525.617,Z 436.584,A -85,B 0,C 180,E1 20898.38,E2 20898.38} C_VEL
LIN {X 0,Y 518.633,Z 426.974,A -85,B 0,C 180,E1 20895.889,E2 20895.889} C_VEL
LIN {X 0,Y 514.668,Z 421.612,A -85,B 0,C 180,E1 20894.284,E2 20894.284} C_VEL
LIN {X 0,Y 510.826,Z 416.479,A -85,B 0,C 180,E1 20892.549,E2 20892.549} C_VEL
LIN {X 0,Y 507.3,Z 411.92,A -85,B 0,C 180,E1 20890.735,E2 20890.735} C_VEL
LIN {X 0,Y 503.745,Z 407.251,A -85,B 0,C 180,E1 20888.561,E2 20888.561} C_VEL
LIN {X 0,Y 499.703,Z 401.937,A -85,B 0,C 180,E1 20885.281,E2 20885.281} C_VEL
LIN {X 0,Y 496.09,Z 397.773,A -85,B 0,C 180,E1 20879.538,E2 20879.538} C_VEL
LIN {X 0,Y 495.997,Z 397.574,A -85,B 0,C 180,E1 20876.764,E2 20876.764} C_VEL
LIN {X 0,Y 497.397,Z 399.754,A -85,B 0,C 180,E1 20873.188,E2 20873.188} C_VEL
LIN {X 0,Y 500.396,Z 402.791,A -85,B 0,C 180,E1 20869.814,E2 20869.814} C_VEL
LIN {X 0,Y 504.917,Z 408.713,A -85,B 0,C 180,E1 20866.428,E2 20866.428} C_VEL
LIN {X 0,Y 509.261,Z 414.395,A -85,B 0,C 180,E1 20863.987,E2 20863.987} C_VEL
LIN {X 0,Y 513.061,Z 419.329,A -85,B 0,C 180,E1 20862.183,E2 20862.183} C_VEL
LIN {X 0,Y 517.538,Z 425.394,A -85,B 0,C 180,E1 20860.297,E2 20860.297} C_VEL
LIN {X 0,Y 522.343,Z 431.974,A -85,B 0,C 180,E1 20858.495,E2 20858.495} C_VEL
LIN {X 0,Y 529.645,Z 442.358,A -85,B 0,C 180,E1 20856.083,E2 20856.083} C_VEL
LIN {X 0,Y 538.256,Z 455.504,A -85,B 0,C 180,E1 20853.582,E2 20853.582} C_VEL
LIN {X 0,Y 544.694,Z 466.036,A -85,B 0,C 180,E1 20851.89,E2 20851.89} C_VEL
LIN {X 0,Y 532.133,Z 673.079,A -85,B 0,C 180,E1 20848.629,E2 20848.629} C_VEL
LIN {X 0,Y 523.655,Z 818.486,A -85,B 0,C 180,E1 20846.334,E2 20846.334} C_VEL
LIN {X 0,Y 520.827,Z 846.19,A -85,B 0,C 180,E1 20845.795,E2 20845.795} C_VEL
LIN {X 0,Y 517.014,Z 872.032,A -85,B 0,C 180,E1 20845.125,E2 20845.125} C_VEL
LIN {X 0,Y 513.399,Z 892.902,A -85,B 0,C 180,E1 20844.447,E2 20844.447} C_VEL
LIN {X 0,Y 509.432,Z 912.862,A -85,B 0,C 180,E1 20843.676,E2 20843.676} C_VEL
LIN {X 0,Y 504.675,Z 934.379,A -85,B 0,C 180,E1 20842.693,E2 20842.693} C_VEL
LIN {X 0,Y 498.386,Z 959.992,A -85,B 0,C 180,E1 20841.298,E2 20841.298} C_VEL
LIN {X 0,Y 492.347,Z 982.056,A -85,B 0,C 180,E1 20839.871,E2 20839.871} C_VEL
LIN {X 0,Y 486.699,Z 1001.482,A -85,B 0,C 180,E1 20838.426,E2 20838.426} C_VEL
LIN {X 0,Y 480.618,Z 1021.48,A -85,B 0,C 180,E1 20836.729,E2 20836.729} C_VEL
LIN {X 0,Y 473.107,Z 1045.185,A -85,B 0,C 180,E1 20834.389,E2 20834.389} C_VEL
LIN {X 0,Y 467.32,Z 1062.896,A -85,B 0,C 180,E1 20832.374,E2 20832.374} C_VEL
LIN {X 0,Y 462.047,Z 1078.948,A -85,B 0,C 180,E1 20830.318,E2 20830.318} C_VEL
LIN {X 0,Y 457.009,Z 1094.452,A -85,B 0,C 180,E1 20828.095,E2 20828.095} C_VEL
LIN {X 0,Y 451.224,Z 1112.63,A -85,B 0,C 180,E1 20825.146,E2 20825.146} C_VEL
LIN {X 0,Y 446.443,Z 1128.196,A -85,B 0,C 180,E1 20822.21,E2 20822.21} C_VEL
LIN {X 0,Y 442.956,Z 1140.365,A -85,B 0,C 180,E1 20819.626,E2 20819.626} C_VEL
LIN {X 0,Y 439.911,Z 1151.821,A -85,B 0,C 180,E1 20816.891,E2 20816.891} C_VEL
LIN {X 0,Y 436.959,Z 1164.53,A -85,B 0,C 180,E1 20813.421,E2 20813.421} C_VEL
LIN {X 0,Y 434.931,Z 1174.506,A -85,B 0,C 180,E1 20810.172,E2 20810.172} C_VEL
LIN {X 0,Y 433.68,Z 1182.041,A -85,B 0,C 180,E1 20807.302,E2 20807.302} C_VEL
LIN {X 0,Y 432.886,Z 1188.107,A -85,B 0,C 180,E1 20804.574,E2 20804.574} C_VEL
LIN {X 0,Y 432.386,Z 1193.073,A -85,B 0,C 180,E1 20801.877,E2 20801.877} C_VEL
LIN {X 0,Y 432.128,Z 1197.017,A -85,B 0,C 180,E1 20799.187,E2 20799.187} C_VEL
LIN {X 0,Y 432.02,Z 1199.945,A -85,B 0,C 180,E1 20796.512,E2 20796.512} C_VEL
LIN {X 0,Y 431.987,Z 1201.875,A -85,B 0,C 180,E1 20793.849,E2 20793.849} C_VEL
LIN {X 0,Y 431.991,Z 1202.792,A -85,B 0,C 180,E1 20791.326,E2 20791.326} C_VEL
LIN {X 0,Y 431.99,Z 1202.824,A -85,B 0,C 180,E1 20788.806,E2 20788.806} C_VEL
LIN {X 0,Y 431.985,Z 1201.969,A -85,B 0,C 180,E1 20786.284,E2 20786.284} C_VEL
LIN {X 0,Y 432.015,Z 1200.106,A -85,B 0,C 180,E1 20783.622,E2 20783.622} C_VEL
LIN {X 0,Y 432.116,Z 1197.25,A -85,B 0,C 180,E1 20780.947,E2 20780.947} C_VEL
LIN {X 0,Y 432.361,Z 1193.386,A -85,B 0,C 180,E1 20778.258,E2 20778.258} C_VEL
LIN {X 0,Y 432.853,Z 1188.494,A -85,B 0,C 180,E1 20775.554,E2 20775.554} C_VEL
LIN {X 0,Y 433.63,Z 1182.541,A -85,B 0,C 180,E1 20772.834,E2 20772.834} C_VEL
LIN {X 0,Y 434.869,Z 1175.117,A -85,B 0,C 180,E1 20769.966,E2 20769.966} C_VEL
LIN {X 0,Y 436.901,Z 1165.142,A -85,B 0,C 180,E1 20766.677,E2 20766.677} C_VEL
LIN {X 0,Y 439.802,Z 1152.698,A -85,B 0,C 180,E1 20763.248,E2 20763.248} C_VEL
LIN {X 0,Y 442.807,Z 1141.238,A -85,B 0,C 180,E1 20760.512,E2 20760.512} C_VEL
LIN {X 0,Y 446.265,Z 1128.992,A -85,B 0,C 180,E1 20757.927,E2 20757.927} C_VEL
LIN {X 0,Y 450.606,Z 1114.334,A -85,B 0,C 180,E1 20755.188,E2 20755.188} C_VEL
LIN {X 0,Y 456.102,Z 1096.423,A -85,B 0,C 180,E1 20752.294,E2 20752.294} C_VEL
LIN {X 0,Y 461.131,Z 1080.163,A -85,B 0,C 180,E1 20749.992,E2 20749.992} C_VEL
